	CheckConnectionMsg : STRING(255);
	PositionMsg : STRING(255);
	PositionCountMsg : STRING(255);
	IdMsg : STRING(255);
	CustomMsg : STRING(255);
	
	{region 'Commands'}
		
	{attribute 'OPC.UA.DA' := '0'}
	_moveAbsPosition     : BOOL;
	{attribute 'OPC.UA.DA' := '0'}
	_jogBackwardPosition : BOOL;
	{attribute 'OPC.UA.DA' := '0'}
	_jogForwardPosition  : BOOL;
	{attribute 'OPC.UA.DA' := '0'}
	_customCmd : BOOL;	
	
	{endregion}
	
	{attribute 'OPC.UA.DA' := '0'}
	_initDevice : BOOL;	
	
	{attribute 'OPC.UA.DA' := '0'}
	_pos : INT;	 
	{attribute 'OPC.UA.DA' := '0'}
	_cmd : STRING;	
	{attribute 'OPC.UA.DA' := '0'}
	_itemScheduler : INT;		
	{attribute 'OPC.UA.DA' := '0'}
	_pulseGenerator : TON;	
			
	{attribute 'OPC.UA.DA' := '0'}
	message : STRING;
	{attribute 'OPC.UA.DA' := '0'}
	_length : INT;
	
END_VAR


IF NOT InitConfigSerialCom THEN
	ConfigureSerialCom();
ELSE
	IF _refSerialCom.ErrorReceiveId = COMERROR_NOERROR THEN
		_refSerialCom(TxBuffer := HardwareGlobalVariables.TxBufferPolarisation, 
		 	      	  RxBuffer := HardwareGlobalVariables.RxBufferPolarisation);
	END_IF	
				  
	// Init device
	InitDevice(); 				  
				  
	// Deliver messages
	IF _refSerialCom.IsReceived THEN
		CASE _deliverMessages OF			
			EFeedbackMsgPolarisationFW212C.CheckConnectionMsg :
				CheckConnectionMsg := _refSerialCom.LastReceivedString;	
			EFeedbackMsgPolarisationFW212C.PositionMsg :
				PositionMsg := _refSerialCom.LastReceivedString;
			EFeedbackMsgPolarisationFW212C.PositionCountMsg :
				PositionCountMsg := _refSerialCom.LastReceivedString;
			EFeedbackMsgPolarisationFW212C.IdMsg :
				IdMsg := _refSerialCom.LastReceivedString;
			EFeedbackMsgPolarisationFW212C.CustomMsg :
				CustomMsg := _refSerialCom.LastReceivedString;						
		END_CASE
		
		_deliverMessages := 0;
	END_IF							   							   		
END_IF

IF InitConfigSerialCom THEN			
	MoveAbsPosition(_moveAbsPosition, _pos);	
	JogBackwardPosition(_jogBackwardPosition);				
	JogForwardPosition(_jogForwardPosition);
	CustomCommand(_customCmd, _cmd);	

	IF (NOT _moveAbsPosition AND NOT _jogBackwardPosition AND NOT _jogForwardPosition AND NOT _customCmd) THEN
		MessageScheduler();
	END_IF	
END_IF

METHOD CheckConnection
VAR_INPUT
END_VAR
VAR
	cmd : STRING := '';
END_VAR
_deliverMessages := EFeedbackMsgPolarisationFW212C.CheckConnectionMsg;
_serialCom.Send(cmd);
END_METHOD

METHOD ConfigureSerialCom
VAR_INPUT
END_VAR
IF _coeAccess.CoeOperation.Ready THEN
	_logger.Information(_message.Reset().Append('Start configuration com serial').ToString());
END_IF;	

_coeAccess.CoeOperation.Start();
_coeAccess(SerialCommunication := _config.SerialCommunication);
	
IF _coeAccess.CoeOperation.Done THEN
	_coeAccess.SetDone();
	
	_Logger.Information(_message.Reset().
							Append('{').Append(TO_STRING(THIS^.Family)).Append('} : ').
							Append(' - Status : ').Append(TO_STRING(_coeAccess.Status)).ToString());	
	InitConfigSerialCom := TRUE;
END_IF
 
IF _coeAccess.CoeOperation.Error THEN	
	_coeAccess.SetError(0);
	
	_Logger.Error(_message.Reset().
							Append('{').Append(TO_STRING(THIS^.Family)).Append('} : ').
							Append(' - Status : ').Append(TO_STRING(_coeAccess.Status)).ToString());	
	InitConfigSerialCom := TRUE;
END_IF

THIS^.Status := _coeAccess.Status;
State := _coeAccess.Status;
END_METHOD

{attribute 'TcRpcEnable' := '1'}
METHOD CustomCommand
VAR_INPUT
	Execute : BOOL;
	Cmd : STRING;
END_VAR
IF Execute THEN
	_logger.Information(_message.Reset().
								Append(_config.Name).
								Append(' - Custom : ').
								Append(Cmd).ToString());	
	_deliverMessages := EFeedbackMsgPolarisationFW212C.CustomMsg;								
	_serialCom.Send(Cmd);
	
	_customCmd := FALSE;
END_IF
END_METHOD

METHOD FB_init : BOOL
VAR_INPUT
	bInitRetains : BOOL; // if TRUE, the retain variables are initialized (warm start / cold start)
	bInCopyCode : BOOL;  // if TRUE, the instance afterwards gets moved into the copy code (online change)
	Config : FW212CPolarisationFilterConfig;
END_VAR
IF Config.IsEnabled THEN
	_config := Config;
	
	SUPER^._polarisationFilterConfig.Name := Config.Name;
	SUPER^._polarisationFilterConfig.DeviceID := Config.DeviceID;
	SUPER^._polarisationFilterConfig.IsEnabled := Config.IsEnabled;
	SUPER^._polarisationFilterConfig.LogLevel := Config.LogLevel;
	
	SUPER^.Name := Config.Name;
	SUPER^.DeviceID := Config.DeviceID;	
	THIS^.Family := DeviceFamily.PolarisationFilter;
	
	_Logger.Information(_message.Reset().Append('Init ').
							Append('{').Append(TO_STRING(THIS^.Family)).Append('} - ').
							Append('{').Append(TO_STRING(Config.Name)).Append('}').ToString());																													
END_IF
END_METHOD

(** Returns the model number and firmware version **)
METHOD GetIdentifier : STRING
VAR_INPUT
END_VAR
VAR
	cmd : STRING := '*idn?';
END_VAR
_deliverMessages := EFeedbackMsgPolarisationFW212C.IdMsg;
_serialCom.Send(cmd);
END_METHOD

(** Position Query **)
METHOD PROTECTED GetPosition 
VAR_INPUT
END_VAR
VAR
	cmd : STRING := 'pos?';
END_VAR
_deliverMessages := EFeedbackMsgPolarisationFW212C.PositionMsg;
_serialCom.Send(cmd);
END_METHOD

(** Returns the wheel type **)
METHOD GetPositionCount
VAR_INPUT
END_VAR
VAR
	cmd : STRING := 'pcount?';
END_VAR
_deliverMessages := EFeedbackMsgPolarisationFW212C.PositionCountMsg;
_serialCom.Send(cmd);
END_METHOD

PROPERTY InitConfigSerialCom : BOOL
GET
InitConfigSerialCom := _initConfigSerialCom;
END_GET
SET
_initConfigSerialCom := InitConfigSerialCom;
END_SET
END_PROPERTY

METHOD InitDevice
VAR_INPUT
END_VAR
IF NOT _initDevice THEN	
	_logger.Information(_message.Reset().
								Append(_config.Name).
								Append(' - Init device').ToString());

	// TODO : define max count 
	
	_initDevice := TRUE;	
END_IF
END_METHOD

{attribute 'TcRpcEnable' := '1'}
(** Decrements the filter position by 1 **)
METHOD PROTECTED JogBackwardPosition
VAR_INPUT
	Execute : BOOL;
END_VAR
VAR
	DecFilterPos : BYTE := 68;
	posArray     : ARRAY[1..3] OF BYTE := [27, 91, DecFilterPos];
END_VAR
IF Execute THEN
	_logger.Information(_message.Reset().
								Append(_config.Name).
								Append(' - Jog backward position').ToString());
	_serialCom.Send3B(posArray);
	_jogBackwardPosition := FALSE;
END_IF
END_METHOD

{attribute 'TcRpcEnable' := '1'}
(** Increments the filter position by 1 **)
METHOD PROTECTED JogForwardPosition
VAR_INPUT
	Execute : BOOL;
END_VAR
VAR
	jogForwardPos : BYTE := 67;
	posArray     : ARRAY[1..3] OF BYTE := [27, 91, jogForwardPos];
END_VAR
IF Execute THEN
	_logger.Information(_message.Reset().
								Append(_config.Name).
								Append(' - Jog forward position').ToString());
	_serialCom.Send3B(posArray);
	_jogForwardPosition := FALSE;
END_IF
END_METHOD

METHOD MessageScheduler
VAR_INPUT
END_VAR
IF _pulseGenerator.Q THEN
	_pulseGenerator(IN := FALSE, PT := T#10MS);
		
	CASE _itemScheduler OF
		0:  GetIdentifier();
			_itemScheduler := 1;

		1:	GetPosition();
			_itemScheduler := 2;
			
		2:  GetPositionCount();
			_itemScheduler := 3;
			
		3:  CheckConnection();
			_itemScheduler := 0;								
	END_CASE
ELSE
	_pulseGenerator(IN := TRUE, PT := T#50MS);	
END_IF
END_METHOD

{attribute 'TcRpcEnable' := '1'}
(** Moves the wheel to filter position n **)
METHOD PROTECTED MoveAbsPosition
VAR_INPUT
	Execute : BOOL;
	Position : LREAL;
END_VAR
VAR
	cmd : STRING := 'pos=';
END_VAR
IF Execute THEN
	_logger.Information(_message.Reset().
								Append(_config.Name).
								Append(' - Move absolute position : ').Append(TO_STRING(Position)).ToString());
	_serialCom.Send(CONCAT(cmd, TO_STRING(Position)));
	_moveAbsPosition := FALSE;
END_IF
END_METHOD

{attribute 'TcRpcEnable' := '1'}
METHOD RaisePropertiesChanged
VAR_INPUT
	Execute : BOOL;
END_VAR
IF Execute THEN
	CheckConnectionMsg := ' ';
	PositionMsg := ' ';
	IdMsg := ' ';
	CustomMsg := ' ';
END_IF
END_METHOD

END_FUNCTION_BLOCK

// ---- PMShared/Hardware/Devices/PolarisationFilters/PolarisationFilterBase.TcPOU
FUNCTION_BLOCK ABSTRACT PolarisationFilterBase EXTENDS TExecution IMPLEMENTS IDevice
VAR_INPUT
END_VAR
VAR_OUTPUT
END_VAR
VAR
	{attribute 'OPC.UA.DA' := '0'}
	_name : STRING;
	{attribute 'OPC.UA.DA' := '0'}
	_deviceID : STRING;					
	{attribute 'OPC.UA.DA' := '0'}
	_family : DeviceFamily;			
	{attribute 'OPC.UA.DA' := '0'}
	_logger : Logger;
	{attribute 'OPC.UA.DA' := '0'}
	_message : StringBuilder;
	{attribute 'OPC.UA.DA' := '0'}
	_polarisationFilterConfig : DeviceConfiguration;
END_VAR

PROPERTY DeviceID : STRING
GET
DeviceID := _deviceID;
END_GET
SET
_deviceID := DeviceID;
END_SET
END_PROPERTY

PROPERTY Family : DeviceFamily
GET
Family := _family;
END_GET
SET
_family := Family;
END_SET
END_PROPERTY

METHOD PROTECTED ABSTRACT GetPosition 
VAR_INPUT
END_VAR
END_METHOD

METHOD PROTECTED ABSTRACT JogBackwardPosition
VAR_INPUT
	Execute : BOOL;
END_VAR
END_METHOD

METHOD PROTECTED ABSTRACT JogForwardPosition
VAR_INPUT
	Execute : BOOL;
END_VAR
END_METHOD

METHOD PROTECTED ABSTRACT MoveAbsPosition
VAR_INPUT
	Execute : BOOL;
	Position : LREAL;
END_VAR
END_METHOD

PROPERTY Name : STRING
GET
Name := _name;
END_GET
SET
_name := Name;
END_SET
END_PROPERTY

END_FUNCTION_BLOCK

// ---- PMShared/Hardware/Devices/PolarisationFilters/Thorlabs/ELL14KPolarisationFilter.TcPOU
{attribute 'OPC.UA.DA' := '1'}
FUNCTION_BLOCK ELL14KPolarisationFilter EXTENDS PolarisationFilterBase
VAR_INPUT
END_VAR
VAR_OUTPUT
END_VAR
VAR
	{attribute 'OPC.UA.DA' := '0'}
	_config : ELL14KPolarisationFilterConfig;
	{attribute 'OPC.UA.DA' := '0'}
	_hsPolarisationConfig : PolarisationConfig;
	{attribute 'OPC.UA.DA' := '0'}
	_htPolarisationConfig : PolarisationConfig;
	{attribute 'OPC.UA.DA' := '0'}
	_coeAccess : CoeAccess;
	{attribute 'OPC.UA.DA' := '0'}
	_initConfigSerialCom : BOOL;	
	{attribute 'OPC.UA.DA' := '0'}
	_serialCom  : SerialCom(Prefix :='', Suffix := Const.CR_LF);
	{attribute 'OPC.UA.DA' := '0'}
	_refSerialCom : REFERENCE TO SerialCom(Prefix :='', Suffix := Const.CR_LF) := _serialCom;	 
	{attribute 'OPC.UA.DA' := '0'}
	_isReceived : BOOL;
	
	{attribute 'OPC.UA.DA' := '0'}
	_deliverMessages : INT;
	
	PositionMsg : STRING(255);
	IdMsg : STRING(255);
	CalibMsg : STRING(255);
	CustomMsg : STRING(255);
	
	{region 'Commands'}	
	
	{attribute 'OPC.UA.DA' := '0'}
	_homePosition 		: BOOL;
	{attribute 'OPC.UA.DA' := '0'}
	_moveAbsPosition	: BOOL;
	{attribute 'OPC.UA.DA' := '0'}
	_moveRelPosition	: BOOL;
	{attribute 'OPC.UA.DA' := '0'}
	_jogBackwardPosition : BOOL;
	{attribute 'OPC.UA.DA' := '0'}
	_jogForwardPosition  : BOOL;
	{attribute 'OPC.UA.DA' := '0'}
	_customCmd : BOOL;
	{attribute 'OPC.UA.DA' := '0'}			  		   
	_raiseProperties : BOOL;
	 		 
	{endregion}
	
	{attribute 'OPC.UA.DA' := '0'}
	_initDevice : BOOL;	
	{attribute 'OPC.UA.DA' := '0'}
	_polarResult : EPolar;
 	
	{attribute 'OPC.UA.DA' := '0'}
	_pos : LREAL;
	{attribute 'OPC.UA.DA' := '0'}
	_cmd : STRING;	
	{attribute 'OPC.UA.DA' := '0'}
	_itemScheduler : INT;	
	{attribute 'OPC.UA.DA' := '0'}
	_itemRaisedProperties : INT;		
	{attribute 'OPC.UA.DA' := '0'}
	_pulseGenerator : TON;	
			
	{attribute 'OPC.UA.DA' := '0'}
	tmpMessage : STRING;
	{attribute 'OPC.UA.DA' := '0'}
	message : STRING;
	{attribute 'OPC.UA.DA' := '0'}
	_length : INT;		 
	{attribute 'OPC.UA.DA' := '0'}
	_findSuffix : INT;
	{attribute 'OPC.UA.DA' := '0'}
	_roundPosition : STRING; 
	{attribute 'OPC.UA.DA' := '0'}
	hsS_temp : STRING;
	{attribute 'OPC.UA.DA' := '0'}
	hsP_temp : STRING;
	{attribute 'OPC.UA.DA' := '0'}
	htS_temp : STRING;
	{attribute 'OPC.UA.DA' := '0'}
	htP_temp : STRING;
	
	_delimeter : STRING := ';';
	{attribute 'OPC.UA.DA' := '0'}
	_firstConcat : STRING;
	{attribute 'OPC.UA.DA' := '0'}
	_secondConcat : STRING;
	{attribute 'OPC.UA.DA' := '0'}
	_thirdConcat : STRING;
	{attribute 'OPC.UA.DA' := '0'}
	_fourthConcat : STRING;
	{attribute 'OPC.UA.DA' := '0'}
	_fithConcat : STRING;
	{attribute 'OPC.UA.DA' := '0'}
	_sixthConcat : STRING;
	
END_VAR


IF NOT InitConfigSerialCom THEN
	ConfigureSerialCom();
ELSIF THIS^.Status = TExecutionState.Ready THEN
	IF _refSerialCom.ErrorReceiveId = COMERROR_NOERROR THEN
		_refSerialCom(TxBuffer:= HardwareGlobalVariables.TxBufferPolarisation, 
		 	          RxBuffer:= HardwareGlobalVariables.RxBufferPolarisation);
	END_IF	
				  
	// Init device
	InitDevice(); 				  
				  
	// Deliver messages
	IF _refSerialCom.IsReceived THEN
		CASE _deliverMessages OF			
			EFeedbackMsgPolarisationELL14K.PositionMsg :
				tmpMessage := DELETE(_refSerialCom.LastReceivedString, 3, 1);
				_length := LEN(tmpMessage);
				_findSuffix := FIND(tmpMessage, Const.CR_LF);
				message := DELETE(tmpMessage, 4, _findSuffix);
				
				PositionMsg := ConvertPulsesToDegrees(message);
				
				_roundPosition := LREAL_TO_FMTSTR(STRING_TO_LREAL(PositionMsg), 1, TRUE);	
				hsS_temp := LREAL_TO_FMTSTR(_hsPolarisationConfig.PolarAngle_S, 1, FALSE); 
				hsP_temp := LREAL_TO_FMTSTR(_hsPolarisationConfig.PolarAngle_P, 1, FALSE);
				htS_temp := LREAL_TO_FMTSTR(_htPolarisationConfig.PolarAngle_S, 1, FALSE); 
				htP_temp := LREAL_TO_FMTSTR(_htPolarisationConfig.PolarAngle_P, 1, FALSE);
				IF (_roundPosition = hsS_temp OR _roundPosition = htS_temp) THEN
					PolarResult := EPolar.S_Polar;
				ELSIF (_roundPosition = hsP_temp OR _roundPosition = htP_temp) THEN
					PolarResult := EPolar.P_Polar;		
				END_IF
								
				_logger.Information(_message.Reset().Append('ELL14KPolarisationFilter position: ').Append(PositionMsg).ToString());
				
			EFeedbackMsgPolarisationELL14K.IdMsg :
				IdMsg := _refSerialCom.LastReceivedString;							
			EFeedbackMsgPolarisationELL14K.CustomMsg :
				CustomMsg := _refSerialCom.LastReceivedString;						
		END_CASE
	ELSE
		CASE _deliverMessages OF
			EFeedbackMsgPolarisationELL14K.CalibMsg :
				_firstConcat := CONCAT(LREAL_TO_FMTSTR(_hsPolarisationConfig.PolarAngle_S, 1, FALSE), _delimeter);	
				_secondConcat := CONCAT(_firstConcat, LREAL_TO_FMTSTR(_hsPolarisationConfig.PolarAngle_P, 1, FALSE));	
				_thirdConcat := CONCAT(_secondConcat, _delimeter);
				_fourthConcat := CONCAT(_thirdConcat, LREAL_TO_FMTSTR(_htPolarisationConfig.PolarAngle_S, 1, FALSE));
				_fithConcat := CONCAT(_fourthConcat, _delimeter);				
				_sixthConcat := CONCAT(_fithConcat, LREAL_TO_FMTSTR(_htPolarisationConfig.PolarAngle_P, 1, FALSE));
			
				CalibMsg := _sixthConcat;
				_deliverMessages := EFeedbackMsgPolarisationELL14K.PositionMsg;
		END_CASE			
	END_IF							   	


	HomePosition(_homePosition);	
	MoveAbsPosition(_moveAbsPosition, _pos);
	MoveRelPosition(_moveRelPosition, _pos);	
	JogBackwardPosition(_jogBackwardPosition);				
	JogForwardPosition(_jogForwardPosition);
	CustomCommand(_customCmd, _cmd);		
	RaisePropertiesChanged(_raiseProperties);		
END_IF

METHOD ConfigureSerialCom
VAR_INPUT
END_VAR
IF _coeAccess.CoeOperation.Ready THEN
	_logger.Information(_message.Reset().Append('Start configuration com serial').ToString());
END_IF;	

_coeAccess.CoeOperation.Start();
_coeAccess(SerialCommunication := _config.SerialCommunication);
	
IF _coeAccess.CoeOperation.Done THEN
	_coeAccess.SetDone();	
 
	_Logger.Information(_message.Reset().
							Append('{').Append(TO_STRING(THIS^.Family)).Append('} : ').
							Append(' - Status : ').Append(TO_STRING(_coeAccess.Status)).ToString());	
	InitConfigSerialCom := TRUE;
END_IF
 
IF _coeAccess.CoeOperation.Error THEN	
	_coeAccess.SetError(0);
	
	_Logger.Error(_message.Reset().
							Append('{').Append(TO_STRING(THIS^.Family)).Append('} : ').
							Append(' - Status : ').Append(TO_STRING(_coeAccess.Status)).ToString());
	InitConfigSerialCom := TRUE;
END_IF

THIS^.Status := _coeAccess.Status;
State := _coeAccess.Status;
END_METHOD

METHOD ConvertDegreesToPulses : STRING
VAR_INPUT
	AnglePosition : LREAL;
END_VAR
VAR
	NumberPulses : DWORD;
END_VAR
NumberPulses := LREAL_TO_DWORD(AnglePosition * Const.PULSES_PER_DEG);	
ConvertDegreesToPulses := DWORD_TO_HEXSTR(NumberPulses, 8, FALSE );
END_METHOD

METHOD ConvertPulsesToDegrees : STRING
VAR_INPUT
	Pulses : STRING;
END_VAR
VAR
	pulsesInHex : STRING; 
	pulsesToDint : DINT;
END_VAR
pulsesInHex := CONCAT('16#', Pulses);
pulsesToDint := STRING_TO_DINT(pulsesInHex);
ConvertPulsesToDegrees := LREAL_TO_FMTSTR(ABS(DINT_TO_LREAL(pulsesToDint) / Const.PULSES_PER_DEG), 4, TRUE);
END_METHOD

{attribute 'TcRpcEnable' := '1'}
METHOD CustomCommand
VAR_INPUT
	Execute : BOOL;
	Cmd : STRING;
END_VAR
IF Execute THEN
	_logger.Information(_message.Reset().
								Append(_config.Name).
								Append(' - Custom : ').
								Append(Cmd).ToString());
	_deliverMessages := EFeedbackMsgPolarisationELL14K.CustomMsg;									
	_serialCom.Send(Cmd);
	
	_customCmd := FALSE;
END_IF
END_METHOD

METHOD FB_init : BOOL
VAR_INPUT
	bInitRetains : BOOL; // if TRUE, the retain variables are initialized (warm start / cold start)
	bInCopyCode : BOOL;  // if TRUE, the instance afterwards gets moved into the copy code (online change)
	Config : ELL14KPolarisationFilterConfig;
	HsPolarisationConfig : PolarisationConfig;
	HtPolarisationConfig : PolarisationConfig;
END_VAR
IF Config.IsEnabled THEN
	_config := Config;
	_hsPolarisationConfig := HsPolarisationConfig;
	_htPolarisationConfig := HtPolarisationConfig;
	
	SUPER^._polarisationFilterConfig.Name := Config.Name;
	SUPER^._polarisationFilterConfig.DeviceID := Config.DeviceID;
	SUPER^._polarisationFilterConfig.IsEnabled := Config.IsEnabled;
	SUPER^._polarisationFilterConfig.LogLevel := Config.LogLevel;
	
	SUPER^.Name := Config.Name;
	SUPER^.DeviceID := Config.DeviceID;	
	THIS^.Family := DeviceFamily.PolarisationFilter;
	
	_Logger.Information(_message.Reset().Append('Init ').
							Append('{').Append(TO_STRING(THIS^.Family)).Append('} - ').
							Append('{').Append(TO_STRING(Config.Name)).Append('}').ToString());																													
END_IF
END_METHOD

METHOD PROTECTED GetCalibConfig
VAR_INPUT
END_VAR
VAR
	
END_VAR
_deliverMessages := EFeedbackMsgPolarisationELL14K.CalibMsg;
END_METHOD

(** Returns the model number and firmware version **)
METHOD GetIdentifier
VAR_INPUT
END_VAR
VAR
	cmd : STRING := '0i1';
END_VAR
_deliverMessages := EFeedbackMsgPolarisationELL14K.IdMsg;	
_serialCom.Send(cmd);
END_METHOD

METHOD PROTECTED GetPosition
VAR_INPUT
END_VAR
VAR
	cmd : STRING := '0gp';
END_VAR
_deliverMessages := EFeedbackMsgPolarisationELL14K.PositionMsg;
_serialCom.Send(cmd);
END_METHOD

{attribute 'TcRpcEnable' := '1'}
METHOD HomePosition
VAR_INPUT
	Execute : BOOL;
END_VAR
VAR
	cmd : STRING := '0ho1';
END_VAR
IF Execute THEN
	_logger.Information(_message.Reset().
								Append(_config.Name).
								Append(' - Home position : ').ToString());
	
	PolarResult := EPolar.Unknown;
	
	_serialCom.Send(cmd);	
	_homePosition := FALSE;
END_IF
END_METHOD

PROPERTY InitConfigSerialCom : BOOL
GET
InitConfigSerialCom := _initConfigSerialCom;
END_GET
SET
_initConfigSerialCom := InitConfigSerialCom;
END_SET
END_PROPERTY

METHOD InitDevice
VAR_INPUT
END_VAR
IF NOT _initDevice THEN	
	_logger.Information(_message.Reset().
								Append(_config.Name).
								Append(' - Init device').ToString());	
	_initDevice := TRUE;
	//_raiseProperties := TRUE;
	
	GetPosition();	
END_IF
END_METHOD

{attribute 'TcRpcEnable' := '1'}
METHOD PROTECTED JogBackwardPosition
VAR_INPUT
	Execute : BOOL;
END_VAR
VAR
	cmd : STRING := '0bw';
END_VAR
IF Execute THEN
	_logger.Information(_message.Reset().
								Append(_config.Name).
								Append(' - Jog backward position : ').ToString());
	_serialCom.Send(cmd);
	
	_jogBackwardPosition := FALSE;
END_IF
END_METHOD

{attribute 'TcRpcEnable' := '1'}
METHOD PROTECTED JogForwardPosition
VAR_INPUT
	Execute : BOOL;
END_VAR
VAR
	cmd : STRING := '0fw';
END_VAR
IF Execute THEN
	_logger.Information(_message.Reset().
								Append(_config.Name).
								Append(' - Jog forward position : ').ToString());
	_serialCom.Send(cmd);
	
	_jogForwardPosition := FALSE;
END_IF
END_METHOD

{attribute 'TcRpcEnable' := '1'}
METHOD PROTECTED MoveAbsPosition 
VAR_INPUT
	Execute : BOOL;
	Position : LREAL;
END_VAR
VAR
	cmd : STRING := '0ma';
END_VAR
IF Execute THEN
	_pos := Position;	

	_logger.Information(_message.Reset().
								Append(_config.Name).
								Append(' - Move absolute position : ').Append(TO_STRING(_pos)).ToString());
		
	PolarResult := EPolar.Unknown;					
								
	_serialCom.Send(CONCAT(cmd, ConvertDegreesToPulses(_pos)));
	_moveAbsPosition := FALSE;	
END_IF
END_METHOD

{attribute 'TcRpcEnable' := '1'}
METHOD PROTECTED MoveRelPosition 
VAR_INPUT
	Execute : BOOL;
	AnglePosition : LREAL;
END_VAR
VAR
	cmd : STRING := '0mr';
END_VAR
IF Execute THEN
	_pos := AnglePosition;	
	_logger.Information(_message.Reset().
								Append(_config.Name).
								Append(' - Move relative position : ').Append(TO_STRING(_pos)).ToString());
	
	PolarResult := EPolar.Unknown;
	
	_serialCom.Send(CONCAT(cmd, ConvertDegreesToPulses(_pos)));	
	_moveRelPosition := FALSE;
END_IF
END_METHOD

PROPERTY PUBLIC PolarResult : EPolar
GET
PolarResult := _polarResult;
END_GET
SET
_polarResult := PolarResult;
END_SET
END_PROPERTY

{attribute 'TcRpcEnable' := '1'}
METHOD RaisePropertiesChanged
VAR_INPUT
	Execute : BOOL;
END_VAR
IF Execute THEN
	IF THIS^.Status <> TExecutionState.Ready THEN	
		_raiseProperties := FALSE;
		RETURN;
	END_IF
	
	_raiseProperties := TRUE;
	
	IF _pulseGenerator.Q THEN
		_pulseGenerator(IN := FALSE, PT := T#10MS);	

		CASE _itemRaisedProperties OF
			0:  PositionMsg := ' ';
				IdMsg := ' ';
				CalibMsg := ' ';
				CustomMsg := ' ';
				
				_itemRaisedProperties := 10;
			
			10:  GetIdentifier();
				_itemRaisedProperties := 11;
				
			11:  GetPosition();
				_itemRaisedProperties := 12;
				
			12: GetCalibConfig();
				_itemRaisedProperties := 20;
			
			20:  _logger.Information(_message.Reset().
								Append(_config.Name).
								Append(' - Polarisation RaisePropertiesChanged').ToString());
				_raiseProperties := FALSE;				
				_itemRaisedProperties := 0;
			
		END_CASE
	ELSE
		_pulseGenerator(IN := TRUE, PT := T#100MS);	
	END_IF
END_IF
END_METHOD

END_FUNCTION_BLOCK

// ---- PMShared/Hardware/Devices/Lasers/Quantum/SMD12Laser.TcPOU
{attribute 'OPC.UA.DA' := '1'}
FUNCTION_BLOCK SMD12Laser EXTENDS LaserBase
VAR_INPUT
END_VAR
VAR_OUTPUT
END_VAR
VAR
	{attribute 'OPC.UA.DA' := '0'}
	_config : SMD12LaserConfig;	
	{attribute 'OPC.UA.DA' := '0'}
	_coeAccess : CoeAccess;	
	{attribute 'OPC.UA.DA' := '0'}
	_initConfigSerialCom : BOOL;	
	{attribute 'OPC.UA.DA' := '0'}
	_serialCom  : SerialCom(Prefix :='', Suffix := Const.CARRIAGE_RETURN);
	{attribute 'OPC.UA.DA' := '0'}
	_refSerialCom : REFERENCE TO SerialCom(Prefix :='', Suffix := Const.CARRIAGE_RETURN) := _serialCom;		 
	{attribute 'OPC.UA.DA' := '0'}
	_isReceived : BOOL;
	
	{attribute 'OPC.UA.DA' := '0'}
	_deliverMessages : INT;
	
	PowerMsg : STRING(255);
	InterlockStatusMsg : STRING(255);
	LaserTemperatureMsg : STRING(255);
	PsuTemperatureMsg : STRING(255);
	IdMsg : STRING(255);
	CustomMsg : STRING(255);
	
	{region 'Commands'}
	
	{attribute 'OPC.UA.DA' := '0'}
	_powerOn : BOOL;
	{attribute 'OPC.UA.DA' := '0'}
	_powerOff : BOOL;
	{attribute 'OPC.UA.DA' := '0'}
	_setPowerCmd : BOOL;
	{attribute 'OPC.UA.DA' := '0'}	 
	_setCurrentCmd : BOOL;
	{attribute 'OPC.UA.DA' := '0'}			 
	_controlModeCmd : BOOL;
	{attribute 'OPC.UA.DA' := '0'}
	_customCmd : BOOL;	
	{attribute 'OPC.UA.DA' := '0'}			  		   
	_raiseProperties : BOOL;
	
	{endregion}			
	
	{attribute 'OPC.UA.DA' := '0'}
	_initDevice : BOOL;	
	 
	{attribute 'OPC.UA.DA' := '0'}
	_cmd : STRING;			
	{attribute 'OPC.UA.DA' := '0'}
	_setpoint : LREAL := 0;
	{attribute 'OPC.UA.DA' := '0'}
	_itemScheduler : INT;
	{attribute 'OPC.UA.DA' := '0'}
	_itemExecScheduler : INT;		
	{attribute 'OPC.UA.DA' := '0'}
	_itemRaisedProperties : INT;			
	{attribute 'OPC.UA.DA' := '0'}
	_pulseGenerator : TON;	
	{attribute 'OPC.UA.DA' := '0'}
	_execPulseGenerator : TON;	
			
	{attribute 'OPC.UA.DA' := '0'}
	message : STRING;
	{attribute 'OPC.UA.DA' := '0'}	
	_length : INT;
	{attribute 'OPC.UA.DA' := '0'}
	_mode : EControlModeSmd12;	
END_VAR

IF NOT InitConfigSerialCom THEN
	ConfigureSerialCom();
ELSIF THIS^.Status = TExecutionState.Ready THEN
	IF _refSerialCom.ErrorReceiveId = COMERROR_NOERROR THEN
		_refSerialCom(TxBuffer:= HardwareGlobalVariables.TxBufferLaser, 
		 	      	  RxBuffer:= HardwareGlobalVariables.RxBufferLaser);
	END_IF				  
	
	// Init device
	InitDevice(); 				  				 

	// Deliver messages
	IF _refSerialCom.IsReceived THEN				 	
		CASE _deliverMessages OF			
			EFeedbackMsgSMD12.PowerMsg :		
				message := DELETE(_refSerialCom.LastReceivedString, 3, 0);
				_length := LEN(message);		
				PowerMsg := DELETE(message, 4, _length-2);		
			EFeedbackMsgSMD12.InterlockStatusMsg :
				message := DELETE(_refSerialCom.LastReceivedString, 2, 0);
				_length := LEN(message);	
				InterlockStatusMsg := DELETE(message, 2, _length);
			EFeedbackMsgSMD12.LaserTemperatureMsg :
				message := DELETE(_refSerialCom.LastReceivedString, 3, 0);
				_length := LEN(message);		
				LaserTemperatureMsg := DELETE(message, 3, _length-1);
			EFeedbackMsgSMD12.PsuTemperatureMsg :
				message := DELETE(_refSerialCom.LastReceivedString, 3, 0);
				_length := LEN(message);		
				PsuTemperatureMsg := DELETE(message, 3, _length-1);
			EFeedbackMsgSMD12.IdMsg :
				message := DELETE(_refSerialCom.LastReceivedString, 3, 0);
				_length := LEN(message);		
				IdMsg := DELETE(message, 2, _length);
			EFeedbackMsgSMD12.CustomMsg :
				message := DELETE(_refSerialCom.LastReceivedString, 2, 0);
				_length := LEN(message);		
				CustomMsg := DELETE(message, 3, _length);
		END_CASE		
	END_IF								   							   	
	
	PowerOn(_powerOn);
	PowerOff(_powerOff);	
	ControlMode(_controlModeCmd, _mode); 
	SetPower(_setPowerCmd, _setpoint);
	SetCurrent(_setCurrentCmd, _setpoint);
	CustomCommand(_customCmd, _cmd);
	RaisePropertiesChanged(_raiseProperties);
	
	IF (NOT _powerOn AND NOT _powerOff AND NOT _controlModeCmd AND NOT _setPowerCmd AND NOT _setCurrentCmd 
		AND NOT _customCmd AND NOT _raiseProperties) THEN
		MessageScheduler();
	END_IF
END_IF

METHOD ConfigureSerialCom
VAR_INPUT
END_VAR
IF _coeAccess.CoeOperation.Ready THEN
	_logger.Information(_message.Reset().Append('Start configuration com serial').ToString());
END_IF;	

_coeAccess.CoeOperation.Start();
_coeAccess(SerialCommunication := _config.SerialCommunication);
	
IF _coeAccess.CoeOperation.Done THEN
	_coeAccess.SetDone();	
	
	_Logger.Information(_message.Reset().
							Append('{').Append(TO_STRING(THIS^.Family)).Append('} : ').
							Append(' - Status : ').Append(TO_STRING(_coeAccess.Status)).ToString());	
	InitConfigSerialCom := TRUE;
END_IF
 
IF _coeAccess.CoeOperation.Error THEN	
	_coeAccess.SetError(0);
	
	_Logger.Error(_message.Reset().
							Append('{').Append(TO_STRING(THIS^.Family)).Append('} : ').
							Append(' - Status : ').Append(TO_STRING(_coeAccess.Status)).ToString());
	InitConfigSerialCom := TRUE;
END_IF

THIS^.Status := _coeAccess.Status;
State := _coeAccess.Status;
END_METHOD

METHOD ControlMode
VAR_INPUT
	Execute : BOOL;
	Mode : EControlModeSmd12;
END_VAR
VAR
	currentModecmd : STRING := 'CONTROL=CURRENT';
	powerModecmd : STRING := 'CONTROL=POWER';
END_VAR
IF Execute THEN
	_logger.Information(_message.Reset().
								Append(_config.Name).
								Append(' - ControlMode : ').Append(TO_STRING(Mode)).ToString());
	
	IF MODE = EControlModeSmd12.CurrentMode THEN
		_serialCom.Send(currentModecmd);
	ELSIF MODE = EControlModeSmd12.PowerMode THEN
		_serialCom.Send(powerModecmd);
	END_IF
	
	_controlModeCmd := FALSE;		
END_IF
END_METHOD

{attribute 'TcRpcEnable' := '1'}
(** Custom command **)
METHOD CustomCommand
VAR_INPUT
	Execute : BOOL;
	Cmd : STRING;
END_VAR
IF Execute THEN
	_logger.Information(_message.Reset().
								Append(_config.Name).
								Append(' - Custom command : ').
								Append(Cmd).ToString());	
	_deliverMessages := EFeedbackMsgSMD12.CustomMsg;														
	_serialCom.Send(Cmd);	
	_customCmd := FALSE;
END_IF
END_METHOD

METHOD FB_init : BOOL
VAR_INPUT
	bInitRetains : BOOL; // if TRUE, the retain variables are initialized (warm start / cold start)
	bInCopyCode : BOOL;  // if TRUE, the instance afterwards gets moved into the copy code (online change)
	Config : SMD12LaserConfig;
END_VAR
IF Config.IsEnabled THEN
	_config := Config;
	
	SUPER^._laserConfig.Name := Config.Name;
	SUPER^._laserConfig.DeviceID := Config.DeviceID;
	SUPER^._laserConfig.IsEnabled := Config.IsEnabled;
	SUPER^._laserConfig.LogLevel := Config.LogLevel;
	
	SUPER^.Name := Config.Name;
	SUPER^.DeviceID := Config.DeviceID;	
	THIS^.Family := DeviceFamily.Laser;
		
	_Logger.Information(_message.Reset().Append('Init ').
							Append('{').Append(TO_STRING(THIS^.Family)).Append('} - ').
							Append('{').Append(TO_STRING(Config.Name)).Append('}').ToString());																													
END_IF
END_METHOD

METHOD GetIdentifier
VAR_INPUT
END_VAR
VAR
	cmd : STRING := 'VERSION?';
END_VAR
_deliverMessages := EFeedbackMsgSMD12.IdMsg;
_serialCom.Send(cmd);
END_METHOD

(** Returns the status of the Interlock **)
METHOD PROTECTED GetInterlockStatus 
VAR_INPUT
END_VAR
VAR
	cmd : STRING := 'STATUS?';
END_VAR
_deliverMessages := EFeedbackMsgSMD12.InterlockStatusMsg;
_serialCom.Send(cmd);
END_METHOD

(** Returns the temperature of the laser head in degrees centigrade **)
METHOD GetLaserTemperature 
VAR_INPUT
END_VAR
VAR
	cmd : STRING := 'LASTEMP?';
END_VAR
_deliverMessages := EFeedbackMsgSMD12.LaserTemperatureMsg;
_serialCom.Send(cmd);
END_METHOD

(** Returns the temperature of the PSU in degrees centigrade **)
METHOD GetPsuTemperature
VAR_INPUT
END_VAR
VAR
	cmd : STRING := 'PSUTEMP?';
END_VAR
_deliverMessages := EFeedbackMsgSMD12.PsuTemperatureMsg;
_serialCom.Send(cmd);
END_METHOD

{attribute 'TcRpcEnable' := '1'}
(** Returns the timers of the laser and PSU:
		PSU Time=#######.#     Total time the system has been powered
		Laser Enabled Time=#######.#     Total time the diodes have been powered
		Laser OperationTime=#######.#    Total time the diodes have been powered >1 A  
**)
METHOD GetTimers : HoursStruct
VAR_INPUT
	Execute : BOOL;
END_VAR
VAR
	cmd : STRING := 'TIMERS?';
END_VAR
IF Execute THEN
	_logger.Information(_message.Reset().
								Append(_config.Name).
								Append(' - GetTimers').ToString());
	_serialCom.Send(cmd);
END_IF
END_METHOD

PROPERTY InitConfigSerialCom : BOOL
GET
InitConfigSerialCom := _initConfigSerialCom;
END_GET
SET
_initConfigSerialCom := InitConfigSerialCom;
END_SET
END_PROPERTY

METHOD InitDevice
VAR_INPUT
END_VAR
IF NOT _initDevice THEN	
	_logger.Information(_message.Reset().
								Append(_config.Name).
								Append(' - InitDevice').ToString());	
	_raiseProperties:= TRUE;	
	_initDevice := TRUE;	
END_IF
END_METHOD

METHOD MessageScheduler
VAR_INPUT
END_VAR
IF _pulseGenerator.Q THEN
	_pulseGenerator(IN := FALSE, PT := T#10MS);
		
	CASE _itemScheduler OF		
		0:	ReadPower();
			_itemScheduler := 1;				
	
		1:  GetLaserTemperature();
			_itemScheduler := 2;	
		
		2:  GetPsuTemperature();
			_itemScheduler := 0;		
	END_CASE
ELSE
	_pulseGenerator(IN := TRUE, PT := T#100MS);		
END_IF
END_METHOD

{attribute 'TcRpcEnable' := '1'}
(** Disables the laser, regardless of the interlock status **)
METHOD PROTECTED PowerOff
VAR_INPUT
	Execute : BOOL;
END_VAR
VAR
	cmd : STRING := 'OFF';
END_VAR
IF Execute THEN	
	_powerOff := TRUE;	
	
	IF _execPulseGenerator.Q THEN
		_execPulseGenerator(IN := FALSE, PT := T#10MS);
			
		CASE _itemExecScheduler OF
			0: _logger.Information(_message.Reset().
								Append(_config.Name).
								Append(' - PowerOff').ToString());
				_serialCom.Send(cmd);
				_itemExecScheduler := 1;
			
			1:  GetInterlockStatus();
				_itemExecScheduler := 2;
				
			2:  _powerOff := FALSE;	
				_itemExecScheduler := 0;		
								
		END_CASE
	ELSE
		_execPulseGenerator(IN := TRUE, PT := T#100MS);	
	END_IF
END_IF
END_METHOD

{attribute 'TcRpcEnable' := '1'}
(* Enables the laser subject to Interlock and Enable Switch status *)
METHOD PROTECTED PowerOn
VAR_INPUT
	Execute : BOOL;
END_VAR
VAR
	cmd : STRING := 'ON';
END_VAR
IF Execute THEN	
	_powerOn := TRUE;	

	IF _execPulseGenerator.Q THEN
		_execPulseGenerator(IN := FALSE, PT := T#10MS);
			
		CASE _itemExecScheduler OF
			0: _logger.Information(_message.Reset().
								Append(_config.Name).
								Append(' - PowerOn').ToString());
				_serialCom.Send(cmd);
				_itemExecScheduler := 1;
			
			1:  GetInterlockStatus();
				_itemExecScheduler := 2;
				
			2:  _powerOn := FALSE;	
				_itemExecScheduler := 0;		
								
		END_CASE
	ELSE
		_execPulseGenerator(IN := TRUE, PT := T#100MS);	
	END_IF
END_IF
END_METHOD

{attribute 'TcRpcEnable' := '1'}
METHOD RaisePropertiesChanged
VAR_INPUT
	Execute : BOOL;
END_VAR
IF Execute THEN
	_raiseProperties := TRUE;
	
	IF _pulseGenerator.Q THEN
		_pulseGenerator(IN := FALSE, PT := T#10MS);	

		CASE _itemRaisedProperties OF
			0:  InterlockStatusMsg := ' ';
				IdMsg := ' ';
				CustomMsg := ' ';
				
				_itemRaisedProperties := 10;
			
			10:  GetIdentifier();
				_itemRaisedProperties := 11;
				
			11:  GetInterlockStatus();
				_itemRaisedProperties := 12;
			
			12:  _logger.Information(_message.Reset().
								Append(_config.Name).
								Append(' - RaisePropertiesChanged').ToString());
				_raiseProperties := FALSE;				
				_itemRaisedProperties := 0;
			
		END_CASE
	ELSE
		_pulseGenerator(IN := TRUE, PT := T#100MS);	
	END_IF
END_IF
END_METHOD

(** Returns the power of the laser **)
METHOD PROTECTED ReadPower 
VAR_INPUT
END_VAR
VAR
	cmd : STRING := 'POWER?';
END_VAR
_deliverMessages := EFeedbackMsgSMD12.PowerMsg;	
_serialCom.Send(cmd);
END_METHOD

{attribute 'TcRpcEnable' := '1'}
METHOD SetCurrent 
VAR_INPUT
	Execute : BOOL;
	Current : LREAL;
END_VAR
VAR
	cmd : STRING := 'CURRENT=';
END_VAR
IF Execute THEN	
	_setCurrentCmd := TRUE;	
	
	_setpoint := Current;

	IF _execPulseGenerator.Q THEN
		_execPulseGenerator(IN := FALSE, PT := T#10MS);
			
		CASE _itemExecScheduler OF
			0: _logger.Information(_message.Reset().
								Append(_config.Name).
								Append(' - SetCurrent : ').Append(TO_STRING(_setpoint)).ToString());
				_serialCom.Send(CONCAT(cmd, TO_STRING(_setpoint)));
				_itemExecScheduler := 1;
			
			1:  _setCurrentCmd := FALSE;	
				_itemExecScheduler := 0;		
								
		END_CASE
	ELSE
		_execPulseGenerator(IN := TRUE, PT := T#100MS);	
	END_IF
END_IF
END_METHOD

{attribute 'TcRpcEnable' := '1'}
(** This sets the output power of the laser 
For example, to set a power of 2800 mW, send the string POWER=2800, followed by striking the RETURN key
**)
METHOD PROTECTED SetPower 
VAR_INPUT
	Execute : BOOL;
	Power : LREAL;
END_VAR
VAR
	cmd : STRING := 'POWER=';
END_VAR
IF Execute THEN	
	_setPowerCmd := TRUE;	

	_setpoint := Power;
	
	IF _execPulseGenerator.Q THEN
		_execPulseGenerator(IN := FALSE, PT := T#10MS);
			
		CASE _itemExecScheduler OF
			0: _logger.Information(_message.Reset().
								Append(_config.Name).
								Append(' - SetPower : ').Append(TO_STRING(_setpoint)).ToString());
				_serialCom.Send(CONCAT(cmd, TO_STRING(_setpoint)));
				_itemExecScheduler := 1;
			
			1:  ReadPower();
				_itemExecScheduler := 2;
				
			2:  _setPowerCmd := FALSE;	
				_itemExecScheduler := 0;		
								
		END_CASE
	ELSE
		_execPulseGenerator(IN := TRUE, PT := T#100MS);	
	END_IF
END_IF
END_METHOD

END_FUNCTION_BLOCK

// ---- PMShared/Hardware/Devices/Lasers/LaserBase.TcPOU
FUNCTION_BLOCK ABSTRACT LaserBase EXTENDS TExecution IMPLEMENTS IDevice
VAR_INPUT
END_VAR
VAR_OUTPUT
END_VAR
VAR
	{attribute 'OPC.UA.DA' := '0'}
	_name : STRING;
	{attribute 'OPC.UA.DA' := '0'}
	_deviceID : STRING;				
	{attribute 'OPC.UA.DA' := '0'}	
	_family : DeviceFamily;	
	{attribute 'OPC.UA.DA' := '0'}
	_logger : Logger;
	{attribute 'OPC.UA.DA' := '0'}
	_message : StringBuilder;
	{attribute 'OPC.UA.DA' := '0'}
	_laserConfig : DeviceConfiguration;	
END_VAR

PROPERTY DeviceID : STRING
GET
DeviceID := _deviceID;
END_GET
SET
_deviceID := DeviceID;
END_SET
END_PROPERTY

PROPERTY Family : DeviceFamily
GET
Family := _family;
END_GET
SET
_family := Family;
END_SET
END_PROPERTY

METHOD PROTECTED ABSTRACT GetInterlockStatus 
VAR_INPUT
END_VAR
END_METHOD

PROPERTY Name : STRING
GET
Name := _name;
END_GET
SET
_name := Name;
END_SET
END_PROPERTY

METHOD PROTECTED ABSTRACT PowerOff
VAR_INPUT
	Execute : BOOL;
END_VAR
END_METHOD

METHOD PROTECTED ABSTRACT PowerOn
VAR_INPUT
	Execute : BOOL;
END_VAR
END_METHOD

METHOD PROTECTED ABSTRACT ReadPower 
VAR_INPUT
END_VAR
END_METHOD

METHOD PROTECTED ABSTRACT SetPower
VAR_INPUT
	Execute : BOOL;
	Power : LREAL;
END_VAR
END_METHOD

END_FUNCTION_BLOCK

// ---- PMShared/Hardware/Devices/Lasers/Coherent/Sapphire488Laser.TcPOU
{attribute 'OPC.UA.DA' := '1'}
FUNCTION_BLOCK Sapphire488Laser EXTENDS LaserBase
VAR_INPUT
END_VAR
VAR_OUTPUT
END_VAR
VAR
	{attribute 'OPC.UA.DA' := '0'}
	_config : Sapphire488LaserConfig;	
	{attribute 'OPC.UA.DA' := '0'}
	_coeAccess : CoeAccess;	
	{attribute 'OPC.UA.DA' := '0'}
	_initConfigSerialCom : BOOL;	
	{attribute 'OPC.UA.DA' := '0'}
	_suffix : STRING := Const.CR_LF;
	{attribute 'OPC.UA.DA' := '0'}
	_serialCom  : SerialCom(Prefix :='', Suffix := _suffix);
	{attribute 'OPC.UA.DA' := '0'}
	_refSerialCom : REFERENCE TO SerialCom(Prefix :='', Suffix := _suffix) := _serialCom;		 
	{attribute 'OPC.UA.DA' := '0'}
	_isReceived : BOOL;
	
	
	{attribute 'OPC.UA.DA' := '0'}
	_deliverMessages : INT;
	
	PowerMsg : STRING(255);
	InterlockStatusMsg : STRING(255);
	BasePlateTemperatureMsg : STRING(255);
	ControllerTemperatureMsg : STRING(255);
	DiodeSetTemperatureMsg : STRING(255);
	MeasuredTemperatureMsg : STRING(255);
	LaserHeadReachedDiodeCurrentLimitMsg : STRING(255);
	IdMsg : STRING(255);
	CustomMsg : STRING(255);
	
	{region 'Commands'}
	
	{attribute 'OPC.UA.DA' := '0'}
	_powerOn : BOOL;
	{attribute 'OPC.UA.DA' := '0'}
	_powerOff : BOOL;
	{attribute 'OPC.UA.DA' := '0'}
	_setPowerCmd : BOOL;
	{attribute 'OPC.UA.DA' := '0'}
	_customCmd : BOOL;	
	{attribute 'OPC.UA.DA' := '0'}			  		   
	_raiseProperties : BOOL;
	
	{endregion}			
	
	{attribute 'OPC.UA.DA' := '0'}
	_initDevice : BOOL;	
	 
	{attribute 'OPC.UA.DA' := '0'}
	_cmd : STRING;			
	{attribute 'OPC.UA.DA' := '0'}
	_setpoint : LREAL := 0;
	{attribute 'OPC.UA.DA' := '0'}
	_itemScheduler : INT;
	{attribute 'OPC.UA.DA' := '0'}
	_itemExecScheduler : INT;		
	{attribute 'OPC.UA.DA' := '0'}
	_itemRaisedProperties : INT;			
	{attribute 'OPC.UA.DA' := '0'}
	_pulseGenerator : TON;	
	{attribute 'OPC.UA.DA' := '0'}
	_execPulseGenerator : TON;	
			
	{attribute 'OPC.UA.DA' := '0'}
	fullMessage : STRING;
	{attribute 'OPC.UA.DA' := '0'}
	message : STRING;
	{attribute 'OPC.UA.DA' := '0'}	
	_length : INT;
	{attribute 'OPC.UA.DA' := '0'}	
	_suffixLength : INT := LEN(_suffix);	
END_VAR

IF NOT InitConfigSerialCom THEN
	ConfigureSerialCom();
ELSIF THIS^.Status = TExecutionState.Ready THEN
	IF _refSerialCom.ErrorReceiveId = COMERROR_NOERROR THEN
		_refSerialCom(TxBuffer:= HardwareGlobalVariables.TxBufferLaser, 
		 	      	  RxBuffer:= HardwareGlobalVariables.RxBufferLaser);
	END_IF				  
	
	// Init device
	IF NOT _initDevice THEN	
		InitDevice(); 		
	ELSE;
		// Deliver messages
		IF _refSerialCom.IsReceived THEN				 
			fullMessage := _refSerialCom.LastReceivedString;
			_length := LEN(fullMessage);
			message := DELETE(fullMessage, _suffixLength, _length-_suffixLength+1);
			
			CASE _deliverMessages OF			
				EFeedbackMsgSapphire488.PowerMsg :	
					PowerMsg := message;		
				EFeedbackMsgSapphire488.InterlockStatusMsg :
					InterlockStatusMsg := message;
				EFeedbackMsgSapphire488.BasePlateTemperatureMsg :
					BasePlateTemperatureMsg := message;
				EFeedbackMsgSapphire488.ControllerTemperatureMsg :
					ControllerTemperatureMsg := message;
				EFeedbackMsgSapphire488.DiodeSetTemperatureMsg :
					DiodeSetTemperatureMsg := message;
				EFeedbackMsgSapphire488.MeasuredTemperatureMsg :
					MeasuredTemperatureMsg := message;
				EFeedbackMsgSapphire488.LaserHeadReachedDiodeCurrentLimitMsg :
					LaserHeadReachedDiodeCurrentLimitMsg := message;
				EFeedbackMsgSapphire488.IdMsg :	
					IdMsg := message;
				EFeedbackMsgSapphire488.CustomMsg :
					CustomMsg := message;
			END_CASE		
		END_IF								   							   	
		
		PowerOn(_powerOn);
		PowerOff(_powerOff);	
		SetPower(_setPowerCmd, _setpoint);
		CustomCommand(_customCmd, _cmd);
		RaisePropertiesChanged(_raiseProperties);
		
		IF (NOT _powerOn AND NOT _powerOff AND NOT _setPowerCmd  
			AND NOT _customCmd AND NOT _raiseProperties) THEN
			MessageScheduler();
		END_IF
	
	END_IF
END_IF

METHOD ConfigureSerialCom
VAR_INPUT
END_VAR
IF _coeAccess.CoeOperation.Ready THEN
	_logger.Information(_message.Reset().Append('Start configuration com serial').ToString());
END_IF;	

_coeAccess.CoeOperation.Start();
_coeAccess(SerialCommunication := _config.SerialCommunication);
	
IF _coeAccess.CoeOperation.Done THEN
	_coeAccess.SetDone();	
	
	_Logger.Information(_message.Reset().
							Append('{').Append(TO_STRING(THIS^.Family)).Append('} : ').
							Append(' - Status : ').Append(TO_STRING(_coeAccess.Status)).ToString());	
	InitConfigSerialCom := TRUE;
END_IF
 
IF _coeAccess.CoeOperation.Error THEN	
	_coeAccess.SetError(0);
	
	_Logger.Error(_message.Reset().
							Append('{').Append(TO_STRING(THIS^.Family)).Append('} : ').
							Append(' - Status : ').Append(TO_STRING(_coeAccess.Status)).ToString());
	InitConfigSerialCom := TRUE;
END_IF

THIS^.Status := _coeAccess.Status;
State := _coeAccess.Status;
END_METHOD

{attribute 'TcRpcEnable' := '1'}
(** Custom command **)
METHOD CustomCommand
VAR_INPUT
	Execute : BOOL;
	Cmd : STRING;
END_VAR
IF Execute THEN
	_logger.Information(_message.Reset().
								Append(_config.Name).
								Append(' - Custom command : ').
								Append(Cmd).ToString());	
	_deliverMessages := EFeedbackMsgSapphire488.CustomMsg;														
	_serialCom.Send(Cmd);	
	_customCmd := FALSE;
END_IF
END_METHOD

METHOD FB_init : BOOL
VAR_INPUT
	bInitRetains : BOOL; // if TRUE, the retain variables are initialized (warm start / cold start)
	bInCopyCode : BOOL;  // if TRUE, the instance afterwards gets moved into the copy code (online change)
	Config : Sapphire488LaserConfig;
END_VAR
IF Config.IsEnabled THEN
	_config := Config;
	
	SUPER^._laserConfig.Name := Config.Name;
	SUPER^._laserConfig.DeviceID := Config.DeviceID;
	SUPER^._laserConfig.IsEnabled := Config.IsEnabled;
	SUPER^._laserConfig.LogLevel := Config.LogLevel;
	
	SUPER^.Name := Config.Name;
	SUPER^.DeviceID := Config.DeviceID;	
	THIS^.Family := DeviceFamily.Laser;
		
	_Logger.Information(_message.Reset().Append('Init ').
							Append('{').Append(TO_STRING(THIS^.Family)).Append('} - ').
							Append('{').Append(TO_STRING(Config.Name)).Append('}').ToString());																													
END_IF
END_METHOD

METHOD GetBasePlateTemperature 
VAR_INPUT
END_VAR
VAR
	cmd : STRING := '?BT';
END_VAR
_deliverMessages := EFeedbackMsgSapphire488.BasePlateTemperatureMsg;
_serialCom.Send(cmd);
END_METHOD

METHOD GetControllerTemperature
VAR_INPUT
END_VAR
VAR
	cmd : STRING := '?PST';
END_VAR
_deliverMessages := EFeedbackMsgSapphire488.ControllerTemperatureMsg;
_serialCom.Send(cmd);
END_METHOD

METHOD GetDiodeSetTemperature 
VAR_INPUT
END_VAR
VAR
	cmd : STRING := '?DST';
END_VAR
_deliverMessages := EFeedbackMsgSapphire488.DiodeSetTemperatureMsg;
_serialCom.Send(cmd);
END_METHOD

METHOD GetIdentifier
VAR_INPUT
END_VAR
VAR
	cmd : STRING := '?SV';
END_VAR
_deliverMessages := EFeedbackMsgSapphire488.IdMsg;
_serialCom.Send(cmd);
END_METHOD

(** Returns the status of the Interlock **)
METHOD PROTECTED GetInterlockStatus 
VAR_INPUT
END_VAR
VAR
	cmd : STRING := '?STA';
END_VAR
_deliverMessages := EFeedbackMsgSapphire488.InterlockStatusMsg;
_serialCom.Send(cmd);
END_METHOD

METHOD GetMeasuredTemperature 
VAR_INPUT
END_VAR
VAR
	cmd : STRING := '?DT';
END_VAR
_deliverMessages := EFeedbackMsgSapphire488.MeasuredTemperatureMsg;
_serialCom.Send(cmd);
END_METHOD

{attribute 'TcRpcEnable' := '1'}
(** Returns the timers of the laser and PSU:
		PSU Time=#######.#     Total time the system has been powered
		Laser Enabled Time=#######.#     Total time the diodes have been powered
		Laser OperationTime=#######.#    Total time the diodes have been powered >1 A  
**)
METHOD GetTimers : HoursStruct
VAR_INPUT
	Execute : BOOL;
END_VAR
VAR
	cmd : STRING := 'TIMERS?';
END_VAR
IF Execute THEN
	_logger.Information(_message.Reset().
								Append(_config.Name).
								Append(' - GetTimers').ToString());
	_serialCom.Send(cmd);
END_IF
END_METHOD

PROPERTY InitConfigSerialCom : BOOL
GET
InitConfigSerialCom := _initConfigSerialCom;
END_GET
SET
_initConfigSerialCom := InitConfigSerialCom;
END_SET
END_PROPERTY

METHOD InitDevice
VAR_INPUT
END_VAR
IF NOT _initDevice THEN	
	IF _pulseGenerator.Q THEN
		_pulseGenerator(IN := FALSE, PT := T#10MS);
			
		CASE _itemScheduler OF		
			0:	_logger.Information(_message.Reset().
								Append(_config.Name).
								Append(' - InitDevice').ToString());	

				_serialCom.Send('>=0'); // Echo off
				_itemScheduler := 1;				
		
			1:  _serialCom.Send('E=1'); // Set echo off
				_itemScheduler := 2;	
			
			2:  _serialCom.Send('T=1');  // Enable automatic servo regulation
				_itemScheduler := 3;	
    	
			3:	_raiseProperties:= TRUE;	
				_initDevice := TRUE;
				_itemScheduler := 0;
		END_CASE
	ELSE
	_pulseGenerator(IN := TRUE, PT := T#500MS);		
	END_IF
END_IF
END_METHOD

(** Returns the temperature of the laser head in degrees centigrade **)
METHOD LaserHeadReachedDiodeCurrentLimit 
VAR_INPUT
END_VAR
VAR
	cmd : STRING := '?MCR';
END_VAR
_deliverMessages := EFeedbackMsgSapphire488.LaserHeadReachedDiodeCurrentLimitMsg;
_serialCom.Send(cmd);
END_METHOD

METHOD MessageScheduler
VAR_INPUT
END_VAR
IF _pulseGenerator.Q THEN
	_pulseGenerator(IN := FALSE, PT := T#10MS);
		
	CASE _itemScheduler OF		
		0:	ReadPower();
			_itemScheduler := 1;				
	
		1:  GetBasePlateTemperature();
			_itemScheduler := 2;	
		
		2:  GetControllerTemperature();
			_itemScheduler := 3;		
			
		3:  GetDiodeSetTemperature();
			_itemScheduler := 4;
			
		4:  GetMeasuredTemperature();
			_itemScheduler := 5;
			
		5:  LaserHeadReachedDiodeCurrentLimit();
			_itemScheduler := 0;	
	END_CASE
ELSE
	_pulseGenerator(IN := TRUE, PT := T#500MS);		
END_IF
END_METHOD

{attribute 'TcRpcEnable' := '1'}
(** Disables the laser, regardless of the interlock status **)
METHOD PROTECTED PowerOff
VAR_INPUT
	Execute : BOOL;
END_VAR
VAR
	cmd : STRING := 'L=0';
END_VAR
IF Execute THEN	
	_powerOff := TRUE;	
	
	IF _execPulseGenerator.Q THEN
		_execPulseGenerator(IN := FALSE, PT := T#10MS);
			
		CASE _itemExecScheduler OF
			0: _logger.Information(_message.Reset().
								Append(_config.Name).
								Append(' - PowerOff').ToString());
				_serialCom.Send(cmd);
				_itemExecScheduler := 1;
			
			1:  GetInterlockStatus();
				_itemExecScheduler := 2;
				
			2:  _powerOff := FALSE;	
				_itemExecScheduler := 0;		
								
		END_CASE
	ELSE
		_execPulseGenerator(IN := TRUE, PT := T#500MS);	
	END_IF
END_IF
END_METHOD

{attribute 'TcRpcEnable' := '1'}
(* Enables the laser subject to Interlock and Enable Switch status *)
METHOD PROTECTED PowerOn
VAR_INPUT
	Execute : BOOL;
END_VAR
VAR
	cmd : STRING := 'L=1';
END_VAR
IF Execute THEN	
	_powerOn := TRUE;	

	IF _execPulseGenerator.Q THEN
		_execPulseGenerator(IN := FALSE, PT := T#10MS);
			
		CASE _itemExecScheduler OF
			0: _logger.Information(_message.Reset().
								Append(_config.Name).
								Append(' - PowerOn').ToString());
				_serialCom.Send(cmd);
				_itemExecScheduler := 1;
			
			1:  GetInterlockStatus();
				_itemExecScheduler := 2;
				
			2:  _powerOn := FALSE;	
				_itemExecScheduler := 0;		
								
		END_CASE
	ELSE
		_execPulseGenerator(IN := TRUE, PT := T#500MS);	
	END_IF
END_IF
END_METHOD

{attribute 'TcRpcEnable' := '1'}
METHOD RaisePropertiesChanged
VAR_INPUT
	Execute : BOOL;
END_VAR
IF Execute THEN
	_raiseProperties := TRUE;
	
	IF _pulseGenerator.Q THEN
		_pulseGenerator(IN := FALSE, PT := T#10MS);	

		CASE _itemRaisedProperties OF
			0:  InterlockStatusMsg := ' ';
				IdMsg := ' ';
				CustomMsg := ' ';
				
				_itemRaisedProperties := 10;
			
			10:  GetIdentifier();
				_itemRaisedProperties := 11;
				
			11:  GetInterlockStatus();
				_itemRaisedProperties := 12;
			
			12:  _logger.Information(_message.Reset().
								Append(_config.Name).
								Append(' - RaisePropertiesChanged').ToString());
				_raiseProperties := FALSE;				
				_itemRaisedProperties := 0;
			
		END_CASE
	ELSE
		_pulseGenerator(IN := TRUE, PT := T#500MS);	
	END_IF
END_IF
END_METHOD

(** Returns the power of the laser **)
METHOD PROTECTED ReadPower 
VAR_INPUT
END_VAR
VAR
	cmd : STRING := '?P';
END_VAR
_deliverMessages := EFeedbackMsgSapphire488.PowerMsg;	
_serialCom.Send(cmd);
END_METHOD

{attribute 'TcRpcEnable' := '1'}
(** This sets the output power of the laser 
For example, to set a power of 2800 mW, send the string POWER=2800, followed by striking the RETURN key
**)
METHOD PROTECTED SetPower 
VAR_INPUT
	Execute : BOOL;
	Power : LREAL;
END_VAR
VAR
	cmd : STRING := 'P=';
END_VAR
IF Execute THEN	
	_setPowerCmd := TRUE;	

	_setpoint := Power;
	
	IF _execPulseGenerator.Q THEN
		_execPulseGenerator(IN := FALSE, PT := T#10MS);
			
		CASE _itemExecScheduler OF
			0: _logger.Information(_message.Reset().
								Append(_config.Name).
								Append(' - SetPower : ').Append(TO_STRING(_setpoint)).ToString());
				_serialCom.Send(CONCAT(cmd, TO_STRING(_setpoint)));
				_itemExecScheduler := 1;
			
			1:  ReadPower();
				_itemExecScheduler := 2;
				
			2:  _setPowerCmd := FALSE;	
				_itemExecScheduler := 0;		
								
		END_CASE
	ELSE
		_execPulseGenerator(IN := TRUE, PT := T#500MS);	
	END_IF
END_IF
END_METHOD

END_FUNCTION_BLOCK

// ---- PMShared/Hardware/Devices/FiberSwitch/Leoni/EOLFiberSwitch.TcPOU
{attribute 'OPC.UA.DA' := '1'}
FUNCTION_BLOCK EOLFiberSwitch EXTENDS FiberSwitchBase
VAR_INPUT
END_VAR
VAR_OUTPUT
END_VAR
VAR
	{attribute 'OPC.UA.DA' := '0'}
	_config : EOLFiberSwitchConfig;
	{attribute 'OPC.UA.DA' := '0'}
	_coeAccess : CoeAccess;
	{attribute 'OPC.UA.DA' := '0'}
	_initConfigSerialCom : BOOL;
	{attribute 'OPC.UA.DA' := '0'}
	_serialCom  : SerialCom(Prefix :='', Suffix := Const.CARRIAGE_RETURN);
	{attribute 'OPC.UA.DA' := '0'}
	_refSerialCom : REFERENCE TO SerialCom(Prefix :='', Suffix := Const.CARRIAGE_RETURN) := _serialCom;	 
	{attribute 'OPC.UA.DA' := '0'}
	_isReceived : BOOL;
	
	{attribute 'OPC.UA.DA' := '0'}
	_deliverMessages : INT;
	
	IdMsg : STRING(255);
	CustomMsg : STRING(255);
	
	{region 'Commands'}
	
	{endregion}
	
	{attribute 'OPC.UA.DA' := '0'}
	_initDevice : BOOL;	
	 
	{attribute 'OPC.UA.DA' := '0'}
	_cmd : STRING;	
	{attribute 'OPC.UA.DA' := '0'}
	_itemScheduler : INT;		
	{attribute 'OPC.UA.DA' := '0'}
	_pulseGenerator : TON;	
			
	{attribute 'OPC.UA.DA' := '0'}
	message : STRING;
	{attribute 'OPC.UA.DA' := '0'}
	_length : INT;
		 
END_VAR


IF NOT InitConfigSerialCom THEN
	ConfigureSerialCom();
ELSE
	_refSerialCom(TxBuffer:= HardwareGlobalVariables.TxBufferFiberSwitch, 
		 	      RxBuffer:= HardwareGlobalVariables.RxBufferFiberSwitch);	
				  
	// Init device
	InitDevice(); 				  				 

	// Deliver messages
	IF _refSerialCom.IsReceived THEN
		_length := LEN(_refSerialCom.LastReceivedString);
		message := DELETE(_refSerialCom.LastReceivedString, 2, _length);
	
		CASE _deliverMessages OF			
			EFeedbackMsgEol.IdMsg :
				IdMsg := message;
			EFeedbackMsgEol.CustomMsg :
				CustomMsg := message;						
		END_CASE
		
		_deliverMessages := 0;
	END_IF					   	
END_IF

IF InitConfigSerialCom THEN	
	MessageScheduler();
END_IF

METHOD ConfigureSerialCom
VAR_INPUT
END_VAR
IF _coeAccess.CoeOperation.Ready THEN
	_logger.Information(_message.Reset().Append('Start configuration com serial').ToString());
END_IF;	

_coeAccess.CoeOperation.Start();
_coeAccess(SerialCommunication := _config.SerialCommunication);
	
IF _coeAccess.CoeOperation.Done THEN
	_coeAccess.SetDone();
	
	_Logger.Information(_message.Reset().
							Append('{').Append(TO_STRING(THIS^.Family)).Append('} : ').
							Append(' - Status : ').Append(TO_STRING(_coeAccess.Status)).ToString());	
	InitConfigSerialCom := TRUE;
END_IF
 
IF _coeAccess.CoeOperation.Error THEN	
	_coeAccess.SetError(0);
	
	_Logger.Error(_message.Reset().
							Append('{').Append(TO_STRING(THIS^.Family)).Append('} : ').
							Append(' - Status : ').Append(TO_STRING(_coeAccess.Status)).ToString());	
	InitConfigSerialCom := TRUE;
END_IF

THIS^.Status := _coeAccess.Status;
END_METHOD

{attribute 'TcRpcEnable' := '1'}
(** Response of the current switch position **)
METHOD PROTECTED CurrentPosition
VAR_INPUT
	Execute : BOOL;
END_VAR
VAR
	cmd : STRING := 'ch?';
END_VAR
IF Execute THEN
	_logger.Information(_message.Reset().
								Append(_config.Name).
								Append(' - CurrentPosition').ToString());
	_serialCom.Send(cmd);
END_IF
END_METHOD

METHOD FB_init : BOOL
VAR_INPUT
	bInitRetains : BOOL; // if TRUE, the retain variables are initialized (warm start / cold start)
	bInCopyCode : BOOL;  // if TRUE, the instance afterwards gets moved into the copy code (online change)
	Config : EOLFiberSwitchConfig;
END_VAR
IF Config.IsEnabled THEN
	_config := Config;
	
	SUPER^._fiberSwitchConfig.Name := Config.Name;
	SUPER^._fiberSwitchConfig.DeviceID := Config.DeviceID;
	SUPER^._fiberSwitchConfig.IsEnabled := Config.IsEnabled;
	SUPER^._fiberSwitchConfig.LogLevel := Config.LogLevel;
	
	SUPER^.Name := Config.Name;
	SUPER^.DeviceID := Config.DeviceID;	
	THIS^.Family := DeviceFamily.FiberSwitch;
		
	_Logger.Information(_message.Reset().Append('Init ').
							Append('{').Append(TO_STRING(THIS^.Family)).Append('} - ').
							Append('{').Append(TO_STRING(Config.Name)).Append('}').ToString());																													
END_IF
END_METHOD

{attribute 'TcRpcEnable' := '1'}
(** Response of the firmware version number **)
METHOD FirmwareVersion
VAR_INPUT
	Execute : BOOL;
END_VAR
VAR
	cmd : STRING := 'firmware?';
END_VAR
IF Execute THEN	
	_logger.Information(_message.Reset().
								Append(_config.Name).
								Append(' - FirmwareVersion').ToString());
	_serialCom.Send(cmd);
END_IF
END_METHOD

PROPERTY InitConfigSerialCom : BOOL
GET
InitConfigSerialCom := _initConfigSerialCom;
END_GET
SET
_initConfigSerialCom := InitConfigSerialCom;
END_SET
END_PROPERTY

METHOD InitDevice
VAR_INPUT
END_VAR
IF NOT _initDevice THEN	
	_logger.Information(_message.Reset().
								Append(_config.Name).
								Append(' - Init device').ToString());

	_initDevice := TRUE;	
END_IF
END_METHOD

METHOD MessageScheduler
VAR_INPUT
END_VAR
IF _pulseGenerator.Q THEN
	_pulseGenerator(IN := FALSE, PT := T#10MS);
		
	CASE _itemScheduler OF
		0:  
			_itemScheduler := 0;					
	END_CASE
ELSE
	_pulseGenerator(IN := TRUE, PT := T#50MS);	
END_IF
END_METHOD

{attribute 'TcRpcEnable' := '1'}
METHOD RaisePropertiesChanged
VAR_INPUT
	Execute : BOOL;
END_VAR
IF Execute THEN	
	IdMsg := ' ';
	CustomMsg := ' ';
END_IF
END_METHOD

{attribute 'TcRpcEnable' := '1'}
(** Sets the switch position **)
METHOD PROTECTED SetSwitchPosition
VAR_INPUT
	Execute : BOOL;
	Position : UINT;
END_VAR
VAR
	cmd : STRING := 'ch';
END_VAR
IF Execute THEN	
	_logger.Information(_message.Reset().
								Append(_config.Name).
								Append(' - SetSwitchPosition : ').Append(TO_STRING(Position)).ToString());
	_serialCom.Send(CONCAT(cmd, TO_STRING(Position)));
	
END_IF
END_METHOD

{attribute 'TcRpcEnable' := '1'}
(** Response of the switch type **)
METHOD SwitchType
VAR_INPUT
	Execute : BOOL;
END_VAR
VAR
	cmd : STRING := 'type?';
END_VAR
IF Execute THEN	
	_logger.Information(_message.Reset().
								Append(_config.Name).
								Append(' - SwitchType').ToString());
	_serialCom.Send(cmd);
END_IF
END_METHOD

END_FUNCTION_BLOCK

// ---- PMShared/Hardware/Devices/FiberSwitch/FiberSwitchBase.TcPOU
FUNCTION_BLOCK ABSTRACT FiberSwitchBase EXTENDS TExecution IMPLEMENTS IDevice
VAR_INPUT
END_VAR
VAR_OUTPUT
END_VAR
VAR
	{attribute 'OPC.UA.DA' := '0'}
	_name : STRING;
	{attribute 'OPC.UA.DA' := '0'}
	_deviceID : STRING;					
	{attribute 'OPC.UA.DA' := '0'}
	_family : DeviceFamily;	
	{attribute 'OPC.UA.DA' := '0'}	
	_logger : Logger;
	{attribute 'OPC.UA.DA' := '0'}
	_message : StringBuilder;
	{attribute 'OPC.UA.DA' := '0'}
	_fiberSwitchConfig : DeviceConfiguration;
END_VAR

METHOD PROTECTED ABSTRACT CurrentPosition
VAR_INPUT
	Execute : BOOL;
END_VAR
END_METHOD

PROPERTY DeviceID : STRING
GET
DeviceID := _deviceID;
END_GET
SET
_deviceID := DeviceID;
END_SET
END_PROPERTY

PROPERTY Family : DeviceFamily
GET
Family := _family;
END_GET
SET
_family := Family;
END_SET
END_PROPERTY

PROPERTY Name : STRING
GET
Name := _name;
END_GET
SET
_name := Name;
END_SET
END_PROPERTY

METHOD PROTECTED ABSTRACT SetSwitchPosition
VAR_INPUT
	Execute : BOOL;
	Position : UINT;
END_VAR
END_METHOD

END_FUNCTION_BLOCK

// ---- PMShared/Hardware/Devices/OpticalPowermeters/Thorlabs/PM101/PM101OpticalPowermeterHs.TcPOU
{attribute 'OPC.UA.DA' := '1'}
FUNCTION_BLOCK PM101OpticalPowermeterHs EXTENDS PM101OpticalPowermeter
VAR_INPUT
END_VAR
VAR_OUTPUT
END_VAR
VAR
	{attribute 'OPC.UA.DA' := '0'}
	_config : PM101OpticalPowermeterConfig;
	{attribute 'OPC.UA.DA' := '0'}
	_polarisationConfig : PolarisationConfig;
	{attribute 'OPC.UA.DA' := '0'}
	_responsivityConfig : ResponsivityConfig;
	{attribute 'OPC.UA.DA' := '0'}
	_rFactorSettings : RFactorSettings;
	{attribute 'OPC.UA.DA' := '0'}
	_coeAccess : CoeAccess;
	{attribute 'OPC.UA.DA' := '0'}
	_initConfigSerialCom : BOOL;
	{attribute 'OPC.UA.DA' := '0'}	
	_serialCom  : SerialCom(Prefix :='', Suffix := Const.LINE_FEED);
	{attribute 'OPC.UA.DA' := '0'}
	_refSerialCom : REFERENCE TO SerialCom(Prefix :='', Suffix := Const.LINE_FEEL) := _serialCom;	
	
	{attribute 'OPC.UA.DA' := '0'}
	_pulseGeneratorInit : TON;	
	{attribute 'OPC.UA.DA' := '0'}
	_itemInit : INT;
END_VAR

IF _config.IsSimulated THEN
	SUPER^(Conf := _config, PolarisationConfig := _polarisationConfig, RFactorSettings := _rfactorSettings, ResponsivityConfig := _responsivityConfig, SerialCom := _serialCom, RefSerialCom := _refSerialCom);
ELSE
	IF NOT InitConfigSerialCom THEN
		ConfigureSerialCom();
	ELSIF THIS^.Status = TExecutionState.Ready THEN
		IF _refSerialCom.ErrorReceiveId = COMERROR_NOERROR THEN
			_refSerialCom(TxBuffer:= HardwareGlobalVariables.TxBufferOpticalPowermeterHs, 
						  RxBuffer:= HardwareGlobalVariables.RxBufferOpticalPowermeterHs);
		END_IF						  			
					
		SUPER^(Conf := _config, PolarisationConfig := _polarisationConfig, RFactorSettings := _rfactorSettings, ResponsivityConfig := _responsivityConfig, SerialCom := _serialCom, RefSerialCom := _refSerialCom);

		// Init device
		InitDevice(); 			
	END_IF
END_IF

METHOD ConfigureSerialCom
VAR_INPUT
END_VAR
IF _coeAccess.CoeOperation.Ready THEN
	_logger.Information(_message.Reset().Append('Start configuration com serial').ToString());
END_IF;	

_coeAccess.CoeOperation.Start();
_coeAccess(SerialCommunication := _config.SerialCommunication);
	
IF _coeAccess.CoeOperation.Done THEN
	_coeAccess.SetDone();
	
	_Logger.Information(_message.Reset().
							Append('{').Append(TO_STRING(THIS^.Family)).Append('} : ').
							Append(' - Status : ').Append(TO_STRING(_coeAccess.Status)).ToString());
	InitConfigSerialCom := TRUE;
END_IF
 
IF _coeAccess.CoeOperation.Error THEN	
	_coeAccess.SetError(0);
	
	_Logger.Error(_message.Reset().
							Append('{').Append(TO_STRING(THIS^.Family)).Append('} : ').
							Append(' - Status : ').Append(TO_STRING(_coeAccess.Status)).ToString());
	InitConfigSerialCom := TRUE;
END_IF

THIS^.Status := _coeAccess.Status;
State := _coeAccess.Status;
END_METHOD

METHOD FB_init : BOOL
VAR_INPUT
	bInitRetains : BOOL; // if TRUE, the retain variables are initialized (warm start / cold start)
	bInCopyCode : BOOL;  // if TRUE, the instance afterwards gets moved into the copy code (online change)
	Config : PM101OpticalPowermeterConfig;
	PolarisationConfig : PolarisationConfig;
	RFactorSettings : RFactorSettings;
	ResponsivityConfig : ResponsivityConfig;
END_VAR
IF Config.IsEnabled THEN
	_config := Config;
	_polarisationConfig := PolarisationConfig;
	_rFactorSettings := RFactorSettings;
	_responsivityConfig := ResponsivityConfig;
	
	SUPER^._opticalPowermeterConfig.Name := Config.Name;
	SUPER^._opticalPowermeterConfig.DeviceID := Config.DeviceID;
	SUPER^._opticalPowermeterConfig.IsEnabled := Config.IsEnabled;
	SUPER^._opticalPowermeterConfig.LogLevel := Config.LogLevel;
	
	SUPER^.Name := Config.Name;
	SUPER^.DeviceID := Config.DeviceID;	
	THIS^.Family := DeviceFamily.OpticalPowermeter;
		
	_Logger.Information(_message.Reset().Append('Init ').
							Append('{').Append(TO_STRING(THIS^.Family)).Append('} - ').
							Append('{').Append(TO_STRING(Config.Name)).Append('}').ToString());																													
END_IF
END_METHOD

PROPERTY InitConfigSerialCom : BOOL
GET
InitConfigSerialCom := _initConfigSerialCom;
END_GET
SET
_initConfigSerialCom := InitConfigSerialCom;
END_SET
END_PROPERTY

METHOD InitDevice 
VAR_INPUT	
END_VAR
IF NOT _initDevice THEN	
	CASE _itemInit OF
		0:  _logger.Information(_message.Reset().Append(_config.Name).Append(' - InitDevice').ToString());
			_itemInit := 1;
		
		1:  SUPER^._rangeAuto := TRUE;
			SUPER^._cmdRange := 'TRUE';
			_itemInit := 2;			
			
		2:  SUPER^._setSensorAttenuation := TRUE;
			SUPER^._cmdSensorAttenuation := _config.Sensor.Attenuation;
			_itemInit := 3;
			
		3:  IF _config.Sensor.Name = Const.POWERMETER_SENSOR_NAME_S150C THEN
				_logger.Error(_message.Reset().Append(_config.Name).Append(' - Sensor name: ').Append(_config.Sensor.Name).ToString());
				_itemInit := 10;
			ELSIF _config.Sensor.Name = Const.POWERMETER_SENSOR_NAME_TAP_COUPLER THEN
				_logger.Error(_message.Reset().Append(_config.Name).Append(' - Sensor name: ').Append(_config.Sensor.Name).ToString());
				_itemInit := 20;
			ELSE
				_logger.Error(_message.Reset().Append(_config.Name).Append(' - NAME OF FAILED SENSOR').ToString());
		    END_IF
			
		10:  SUPER^._setWavelength := TRUE;
			 SUPER^._cmdWavelength := _config.Sensor.Wavelength;
			 _itemInit := 50;		
		
		20:  GetResponsivity();
			 _itemInit := 21;
			
		21:	 _pulseGeneratorInit(IN := TRUE, PT := T#3000MS);
			 IF _pulseGeneratorInit.Q THEN
				_pulseGeneratorInit(IN := FALSE);				
			 	_itemInit := 22;
			 END_IF
		
		22:	 IF ResponsivityMsg = LREAL_TO_STRING(_responsivityConfig.Responsivity_mA_W) THEN
			 	_logger.Information(_message.Reset().Append(_config.Name).Append(' - Responsivity already defined').ToString());
			 	_itemInit := 50;
			 ELSE				 
				_itemInit := 23;
			 END_IF	
			 
		23:  _logger.Information(_message.Reset().
							Append(_config.Name).
							Append(' - Init responsivity: ').
							Append(LREAL_TO_STRING(_responsivityConfig.Responsivity_mA_W)).ToString());
			
			SUPER^._setpoint := _responsivityConfig.Responsivity_ma_W;
			SUPER^._setResponsivity := TRUE;
			
			_itemInit := 50;

		50: _logger.Information(_message.Reset().
							Append(_config.Name).
							Append(' - InitDevice done').ToString());				
			_initDevice	:= TRUE;
	END_CASE			
END_IF
END_METHOD

END_FUNCTION_BLOCK

// ---- PMShared/Hardware/Devices/OpticalPowermeters/Thorlabs/PM101OpticalPowermeter.TcPOU
{attribute 'OPC.UA.DA' := '1'}
FUNCTION_BLOCK PM101OpticalPowermeter EXTENDS OpticalPowermeterBase
VAR_INPUT
	{attribute 'OPC.UA.DA' := '0'}
	Conf : PM101OpticalPowermeterConfig;
	{attribute 'OPC.UA.DA' := '0'}
	PolarisationConfig : PolarisationConfig;
	{attribute 'OPC.UA.DA' := '0'}
	RFactorSettings : RFactorSettings;
	{attribute 'OPC.UA.DA' := '0'}
	ResponsivityConfig : ResponsivityConfig;	
	{attribute 'OPC.UA.DA' := '0'}	
	SerialCom  : SerialCom(Prefix :='', Suffix := Const.LINE_FEED); 
	{attribute 'OPC.UA.DA' := '0'}
	RefSerialCom : REFERENCE TO SerialCom(Prefix :='', Suffix := Const.LINE_FEED) := SerialCom; 
	{attribute 'OPC.UA.DA' := '0'}
	PolarResult : EPolar;	 
END_VAR
VAR_OUTPUT
END_VAR
VAR
	{attribute 'OPC.UA.DA' := '0'}
	IoControlPM101 : IoControlPM101;	

	{attribute 'OPC.UA.DA' := '0'}
	_deliverMessages : INT;
		
	PowerMsg : STRING(255);
	CurrentMsg : STRING(255);		
	IdentifierMsg : STRING(255);
	ResponsivityMsg : STRING(255) := 'Undefined';
	DarkOffsetMsg : STRING(255);
	DarkAdjustStateMsg : STRING(255);
	CustomMsg : STRING(255);	
	SensorTypeMsg : STRING(255);			
	WavelengthMsg : STRING(255);				
	(* Not necessary *)
	BeamDiameterMsg : STRING(255);
	SensorAttenuationMsg : STRING(255);			
	MaxPowerMsg : STRING(255);
	MinPowerMsg : STRING(255);
	WavelengthRangeMsg : STRING(255);	
	CalibMsg : STRING(255);
	
	
	{attribute 'OPC.UA.DA' := '0'}
	_flow : STRING;
	{attribute 'OPC.UA.DA' := '0'}
	_powerRawAbs : LREAL;
	{attribute 'OPC.UA.DA' := '0'}
	_powerCal_mW : LREAL;	
	{attribute 'OPC.UA.DA' := '0'}
	_powerRaw_mW : LREAL;
	{attribute 'OPC.UA.DA' := '0'}
	_current_mA : LREAL;
	{attribute 'OPC.UA.DA' := '0'}
	_darkAdjustState : STRING(255);
	{attribute 'OPC.UA.DA' := '0'}	
	_darkOffset_mW : LREAL;
	{attribute 'OPC.UA.DA' := '0'}	
	_responsivity_mW_mA : LREAL;
	{attribute 'OPC.UA.DA' := '0'}
	_rfactor : LREAL := -1;
	
	{region 'Commands'}
	
	{attribute 'OPC.UA.DA' := '0'}		 
	_abortCmd : BOOL;
	{attribute 'OPC.UA.DA' := '0'}	
	_customCmd : BOOL;	
	{attribute 'OPC.UA.DA' := '0'}
	_setBeamDiameter : BOOL;	
	{attribute 'OPC.UA.DA' := '0'}
	_setWavelength : BOOL;	
	{attribute 'OPC.UA.DA' := '0'}
	 _rangeAuto : BOOL;
	{attribute 'OPC.UA.DA' := '0'}	  
	_setSensorAttenuation : BOOL;
	{attribute 'OPC.UA.DA' := '0'} 		
	_setSensorType : BOOL;	 	
	{attribute 'OPC.UA.DA' := '0'}			  		   
	_raiseProperties : BOOL;
	{attribute 'OPC.UA.DA' := '0'}
	_rangeVariation : BOOL;
	{attribute 'OPC.UA.DA' := '0'}
	_startDarkAdjust : BOOL;	 
	{attribute 'OPC.UA.DA' := '0'}
	_cancelDarkAdjust : BOOL;	
	{attribute 'OPC.UA.DA' := '0'}
	_setResponsivity : BOOL; 
	{endregion}
	
	{attribute 'OPC.UA.DA' := '0'}
	_initDevice : BOOL;	
	{attribute 'OPC.UA.DA' := '0'}
	_monitoringMessages : BOOL;	
	 
	{attribute 'OPC.UA.DA' := '0'}
	_cmd : STRING;
	{attribute 'OPC.UA.DA' := '0'}
	_cmdRange : STRING;
	{attribute 'OPC.UA.DA' := '0'}
	_cmdRangesVariation : STRING;
	{attribute 'OPC.UA.DA' := '0'}
	_cmdBeamDiameter : UINT;
	{attribute 'OPC.UA.DA' := '0'}
	_cmdWavelength : UINT;	
	{attribute 'OPC.UA.DA' := '0'}
	_cmdSensorAttenuation : UINT;	
	{attribute 'OPC.UA.DA' := '0'}
	_cmdSensorType : STRING;
	{attribute 'OPC.UA.DA' := '0'}
	_setpoint : LREAL := 0;
	{attribute 'OPC.UA.DA' := '0'}
	_itemScheduler : INT;
	{attribute 'OPC.UA.DA' := '0'}
	_itemExecScheduler : INT;
	{attribute 'OPC.UA.DA' := '0'}
	_itemRaisedProperties : INT;	
	{attribute 'OPC.UA.DA' := '0'}
	_itemSchedulerResponsivity : INT;	
	{attribute 'OPC.UA.DA' := '0'}
	_pulseGenerator : TON;
	{attribute 'OPC.UA.DA' := '0'}
	_pulseGeneratorMsg : TON;
	{attribute 'OPC.UA.DA' := '0'}
	_pulseGeneratorCmd : TON;
	{attribute 'OPC.UA.DA' := '0'}
	_execPulseGenerator : TON;	
	{attribute 'OPC.UA.DA' := '0'}
	_pulseGeneratorCustom : TON;		
	
	{attribute 'OPC.UA.DA' := '0'}
	message : STRING;
	{attribute 'OPC.UA.DA' := '0'}
	_length : INT;
		
	{attribute 'OPC.UA.DA' := '0'}
	_illumFlow : STRING := ' ';
	{attribute 'OPC.UA.DA' := '0'}
	_delimeter : STRING := ';';
	{attribute 'OPC.UA.DA' := '0'}
	_firstConcat : STRING;
	{attribute 'OPC.UA.DA' := '0'}
	_secondConcat : STRING;
	{attribute 'OPC.UA.DA' := '0'}
	_thirdConcat : STRING;
	{attribute 'OPC.UA.DA' := '0'}
	_fourthConcat : STRING;
	{attribute 'OPC.UA.DA' := '0'}
	_fifthConcat : STRING;
	{attribute 'OPC.UA.DA' := '0'}
	_sixthConcat : STRING;
	{attribute 'OPC.UA.DA' := '0'}
	_seventhConcat : STRING;
END_VAR

IF _illumFlow = ' ' THEN	
	IF (Conf.DeviceID = TO_STRING(EPowerIlluminationFlow.HS)) THEN
		_flow := TO_STRING(EPowerIlluminationFlow.HS);
	ELSE
		_flow := TO_STRING(EPowerIlluminationFlow.HT);
	END_IF	
		
	_illumFlow := CONCAT(_flow, _delimeter);
END_IF		


// Deliver messages
IF RefSerialCom.IsReceived OR Conf.IsSimulated THEN					
	IF NOT Conf.IsSimulated THEN
		_length := LEN(RefSerialCom.LastReceivedString);
		message := DELETE(RefSerialCom.LastReceivedString, 2, _length);
	END_IF
		
	IF _monitoringMessages THEN
		CASE _deliverMessages OF			
			EFeedbackMsgPM101.PowerMsg :
				
				IF PolarResult = EPolar.S_Polar THEN
					_rfactor := RFactorSettings.RFactor_S;
				ELSIF PolarResult = EPolar.P_Polar THEN
					_rfactor := RFactorSettings.RFactor_P;
				END_IF			
				
				_powerRawAbs := ABS(STRING_TO_LREAL(message));
				IF  _powerRawAbs > 0 THEN						
					_powerRaw_mW := _powerRawAbs * 1000;
					_powerCal_mW := _powerRawAbs * 1000 / _rfactor;
					
					_firstConcat := CONCAT(_illumFlow, TO_STRING(_powerRaw_mW));	
					_secondConcat := CONCAT(_firstConcat, _delimeter);	
					_thirdConcat := CONCAT(_secondConcat, TO_STRING(_powerCal_mW));
					_fourthConcat := CONCAT(_thirdConcat, _delimeter);
					
					PowerMsg :=  CONCAT(_fourthConcat, TO_STRING(_rfactor));
				END_IF
			EFeedbackMsgPM101.CurrentMsg :				
				_current_mA := STRING_TO_LREAL(message) * 1000;		
				CurrentMsg := CONCAT(_illumFlow, TO_STRING(_current_mA));	
		END_CASE
	ELSE
		CASE _deliverMessages OF
			EFeedbackMsgPM101.IdentifierMsg :				   		
				IdentifierMsg := CONCAT(_illumFlow, message);
				_logger.Information(_message.Reset().Append('IdentifierMsg: ').Append(IdentifierMsg).ToString());													
			EFeedbackMsgPM101.ResponsivityMsg :			
				_responsivity_mW_mA := (STRING_TO_LREAL(message) * 1E3);		
				ResponsivityMsg := CONCAT(_illumFlow, TO_STRING(_responsivity_mW_mA));	
				_logger.Information(_message.Reset().Append('ResponsivityMsg: ').Append(ResponsivityMsg).ToString());						
				message := ' ';	
				
			EFeedbackMsgPM101.DarkOffsetMsg :						
				_darkOffset_mW := (STRING_TO_LREAL(message) * 1E12); 			
				DarkOffsetMsg := CONCAT(_illumFlow, TO_STRING(_darkOffset_mW));	
				_logger.Information(_message.Reset().Append('DarkOffsetMsg: ').Append(DarkOffsetMsg).ToString());	
			EFeedbackMsgPM101.DarkAdjustStateMsg :				
				DarkAdjustStateMsg := CONCAT(_illumFlow, message);			
				_logger.Information(_message.Reset().Append('DarkAdjustStateMsg: ').Append(DarkAdjustStateMsg).ToString());	
									
			EFeedbackMsgPM101.CustomMsg :		    	
				CustomMsg := CONCAT(_illumFlow, message);	
				_logger.Information(_message.Reset().Append('CustomMsg: ').Append(CustomMsg).ToString());
				
				
			EFeedbackMsgPM101.SensorTypeMsg :				
				SensorTypeMsg := CONCAT(_illumFlow, message);					
			EFeedbackMsgPM101.WavelengthMsg :			
				WavelengthMsg := CONCAT(_illumFlow, message);
			EFeedbackMsgPM101.BeamDiameterMsg :			
				BeamDiameterMsg := CONCAT(_illumFlow, message);			
			EFeedbackMsgPM101.SensorAttenuationMsg :			
				SensorAttenuationMsg := CONCAT(_illumFlow, message);	
			EFeedbackMsgPM101.WavelengthRangeMsg :
				WavelengthRangeMsg := CONCAT(_illumFlow, message);	
			EFeedbackMsgPM101.MaxPowerMsg :
				MaxPowerMsg := CONCAT(_illumFlow, message);
			EFeedbackMsgPM101.MinPowerMsg :
				MinPowerMsg := CONCAT(_illumFlow, message);	
		END_CASE
	END_IF							
	
ELSE
	CASE _deliverMessages OF
		EFeedbackMsgPM101.CalibMsg :				
			_fifthConcat := CONCAT(_illumFlow, LREAL_TO_FMTSTR(RFactorSettings.RFactor_S, 10, TRUE));	
			_sixthConcat := CONCAT(_fifthConcat, _delimeter);
			_seventhConcat := CONCAT(_sixthConcat, LREAL_TO_FMTSTR(RFactorSettings.RFactor_P, 10, TRUE));	
		
			CalibMsg := _seventhConcat;
	END_CASE	
END_IF

// Commands
EnableAutoRange(_rangeAuto, STRING_TO_BOOL(_cmdRange));
RangesVariation(_rangeVariation, _cmdRangesVariation);
StartDarkAdjust(_startDarkAdjust);
CancelDarkAdjust(_cancelDarkAdjust);
Abort(_abortCmd);
RaisePropertiesChanged(_raiseProperties);
CustomCommand(_customCmd, _cmd);

// For init sensor
SetResponsivity(_setResponsivity, _setpoint);
SetBeamDiameter(_setBeamDiameter, _cmdBeamDiameter);
SetWavelength(_setWavelength, _cmdWavelength);
SetSensorAttenuation(_setSensorAttenuation, _cmdSensorAttenuation);
SetSensorType(_setSensorType, _cmdSensorType);

// Monitoring some values 
IF _monitoringMessages THEN
	MessageScheduler();
END_IF

(*
IF (NOT _setBeamDiameter AND NOT _setWavelength AND NOT _rangeAuto AND NOT _setSensorAttenuation
    AND NOT _setSensorType AND NOT _setResponsivity AND NOT _customCmd AND NOT _raiseProperties 
	AND NOT _rangeVariation AND NOT _startDarkAdjust AND NOT _cancelDarkAdjust AND NOT _abortCmd) THEN
	MessageScheduler();
END_IF	
*)

METHOD Abort : BOOL;
VAR_INPUT
	Execute : BOOL;
END_VAR
VAR_OUTPUT
	Stop : BOOL;
END_VAR
VAR
	cmd : STRING := 'ABORt';
END_VAR
IF Execute THEN
	_logger.Information(_message.Reset().
								Append(Conf.Name).
								Append(' - Abort command').ToString());																
	SerialCom.Send(Cmd);	
	_abortCmd := FALSE;
	
	//ABORT := TRUE;		 
END_IF
END_METHOD

{attribute 'TcRpcEnable' := '1'}
METHOD CancelDarkAdjust
VAR_INPUT
	Execute : BOOL;
END_VAR
VAR	
	cmd : STRING := 'Sense:CORRection:COLLect:ZERO:ABORt';	
END_VAR
IF Execute THEN
	_logger.Information(_message.Reset().
								Append(Conf.Name).
								Append(' - Cancel dark adjust').ToString());
	
	//Abort(_abortCmd);
	SerialCom.Send(cmd);
	_cancelDarkAdjust := FALSE;
END_IF
END_METHOD

{attribute 'TcRpcEnable' := '1'}
(** Custom command **)
METHOD CustomCommand
VAR_INPUT
	Execute : BOOL;
	Cmd : STRING;
END_VAR
IF Execute THEN
	_logger.Information(_message.Reset().
								Append(Conf.Name).
								Append(' - Custom command:').
								Append(Cmd).ToString());
	
	_deliverMessages := EFeedbackMsgPM101.CustomMsg;																								
	SerialCom.Send(Cmd);	
	_customCmd := FALSE;
END_IF

(*
IF Execute THEN
	IF _pulseGeneratorCustom.Q THEN
		_pulseGeneratorCustom(IN := FALSE);									
		_customCmd := FALSE;
	ELSE	
		_pulseGeneratorCustom(IN := Execute, PT := T#100MS);										
	END_IF	
END_IF	
*)
END_METHOD

{attribute 'TcRpcEnable' := '1'}
(** Switches the auto-ranging function on and off **)
METHOD EnableAutoRange
VAR_INPUT
	Execute : BOOL;
	Activate : BOOL;
END_VAR
VAR
	cmd : STRING := 'Sense:Power:Dc:Range:AUTO ';
	autorRange : STRING;
END_VAR
IF Execute THEN
	_logger.Information(_message.Reset().
								Append(Conf.Name).
								Append(' - Switches the auto-ranging: ').
								Append(TO_STRING(Activate)).ToString());
	
	IF Activate THEN
		autorRange := 'Sense:Power:Dc:Range:AUTO ON';
	ELSE
		autorRange := 'Sense:Power:Dc:Range:AUTO OFF';
	END_IF
					
	SerialCom.Send(CONCAT(cmd, TO_STRING(Activate)));	
	_rangeAuto := FALSE;
END_IF
END_METHOD

METHOD GetBeamDiameter
VAR_INPUT
END_VAR
VAR	
	cmd : STRING := 'Sense:Correction:beamdiameter? ';	
END_VAR
_logger.Information(_message.Reset().Append('GetBeamDiameter').ToString());
_deliverMessages := EFeedbackMsgPM101.BeamDiameterMsg;

IF NOT Conf.IsSimulated THEN
	SerialCom.Send(cmd);
ELSE
	message := '5';
END_IF
END_METHOD

(** Read the unit’s identification string **)
METHOD GetCalibConfig
VAR_INPUT
END_VAR
VAR
END_VAR
_deliverMessages := EFeedbackMsgPM101.CalibMsg;
END_METHOD

METHOD GetDarkAdjustState
VAR_INPUT
END_VAR
VAR	
	cmd : STRING := 'Sense:Correction:COLLect:ZERO:STATe?';	
END_VAR
_deliverMessages := EFeedbackMsgPM101.DarkAdjustStateMsg;					

IF NOT Conf.IsSimulated THEN
	SerialCom.Send(cmd);
ELSE
	message := 'Simu_ok';
END_IF
END_METHOD

METHOD GetDarkOffset
VAR_INPUT
END_VAR
VAR	
	cmd : STRING := 'Sense:CORRection:COLLect:ZERO:MAGNitude?';	
END_VAR
_deliverMessages := EFeedbackMsgPM101.DarkOffsetMsg;
SerialCom.Send(cmd);
END_METHOD

(** Read the unit’s identification string **)
METHOD GetIdentifier
VAR_INPUT
END_VAR
VAR
	cmd : STRING := 'System:Sensor:IDN?';
END_VAR
_deliverMessages := EFeedbackMsgPM101.IdentifierMsg;
SerialCom.Send(cmd);
END_METHOD

(** Get max measure power **)
METHOD GetMaxPower
VAR_INPUT
END_VAR
VAR	
	cmd : STRING := 'Measure:Scalar:POWer? MAXimum';	
END_VAR
_deliverMessages := EFeedbackMsgPM101.MaxPowerMsg;					
SerialCom.Send(cmd);
END_METHOD

(** Get in measure power **)
METHOD GetMinPower
VAR_INPUT
END_VAR
VAR	
	cmd : STRING := 'Measure:Scalar:POWer? MINimum';	
END_VAR
_deliverMessages := EFeedbackMsgPM101.MinPowerMsg;	
SerialCom.Send(cmd);
END_METHOD

METHOD GetResponsivity
VAR_INPUT
END_VAR
VAR	
	cmd : STRING := 'Sense:Correction:power:pdiode:response?';	
END_VAR
_deliverMessages := EFeedbackMsgPM101.ResponsivityMsg;

IF Conf.IsSimulated THEN
	message := LREAL_TO_STRING(0.05);
ELSE
	SerialCom.Send(cmd);	
END_IF
END_METHOD

(** Get the beam diameter in mm **)
METHOD GetSensorAttenuation
VAR_INPUT
END_VAR
VAR	
	cmd : STRING := 'Sense:Correction:BEAMdiameter? ';	
END_VAR
//_logger.Information(_message.Reset().Append('GetSensorAttenuation').ToString());
_deliverMessages := EFeedbackMsgPM101.SensorAttenuationMsg;

IF NOT Conf.IsSimulated THEN
	SerialCom.Send(cmd);
ELSE
	message := INT_TO_STRING(2);
END_IF
END_METHOD

METHOD GetSensorType
VAR_INPUT
END_VAR
VAR	
	cmd : STRING := 'Input:Adapter:TYPE?';	
END_VAR
//_logger.Information(_message.Reset().Append('GetSensorType').ToString());
_deliverMessages := EFeedbackMsgPM101.SensorTypeMsg;

IF Conf.IsSimulated THEN
	message := 'SIMU_PHOTODIODE';	
ELSE
	SerialCom.Send(cmd);
END_IF



(*IF _pulseGeneratorCmd.Q THEN
	_pulseGeneratorCmd(IN := FALSE, PT := T#10MS);	
								
	SerialCom.Send(cmd);
ELSE
	_deliverMessages := EFeedbackMsgPM101.SensorTypeMsg;
	_pulseGeneratorCmd(IN := TRUE, PT := T#100MS);										
END_IF	*)
END_METHOD

(** Get wavelength **)
METHOD GetWavelength
VAR_INPUT
END_VAR
VAR	
	cmd : STRING := 'Sense:CORR:WAVE?';	
END_VAR
_deliverMessages := EFeedbackMsgPM101.WavelengthMsg;

IF Conf.IsSimulated THEN
	message := INT_TO_STRING(473);
ELSE	
	SerialCom.Send(cmd);
END_IF	


(*IF _pulseGeneratorCmd.Q THEN
	_pulseGeneratorCmd(IN := FALSE, PT := T#10MS);	
								
	SerialCom.Send(cmd);
ELSE
	_deliverMessages := EFeedbackMsgPM101.WavelengthMsg;
	_pulseGeneratorCmd(IN := TRUE, PT := T#100MS);										
END_IF*)
END_METHOD

(** Get wavelength range **)
METHOD GetWavelengthRange
VAR_INPUT
END_VAR
VAR	
	cmd : STRING := 'Sense:Power:Dc:Range:UPPer? MINimum ';	
END_VAR
_deliverMessages := EFeedbackMsgPM101.WavelengthRangeMsg;
SerialCom.Send(cmd);
END_METHOD

METHOD MessageScheduler
VAR_INPUT
END_VAR
IF _pulseGenerator.Q THEN
	_pulseGenerator(IN := FALSE, PT := T#10MS);
		
	CASE _itemScheduler OF		   
		0:	ReadPower();	
			_itemScheduler := 1;
			
		1: ReadCurrent();			
		   _itemScheduler := 0;
	END_CASE
ELSE
	_pulseGenerator(IN := TRUE, PT := T#50MS);	
END_IF


(*CASE _itemScheduler OF
	0:  _pulseGeneratorMsg(IN := TRUE, PT := T#10MS); // 50MS + 10MS de temps de cycle = 60 MS 
		IF _pulseGeneratorMsg.Q THEN
			_pulseGeneratorMsg(IN := FALSE);			
			
			ReadPower();			
			_itemScheduler := 1;
		END_IF 

	1:  _pulseGeneratorMsg(IN := TRUE, PT := T#100MS); // 50MS + 10MS de temps de cycle = 60 MS 
		IF _pulseGeneratorMsg.Q THEN
			_pulseGeneratorMsg(IN := FALSE);			
			
			ReadCurrent();			
			_itemScheduler := 0;
		END_IF  												
END_CASE
*)
END_METHOD

{attribute 'TcRpcEnable' := '1'}
METHOD RaisePropertiesChanged
VAR_INPUT
	Execute : BOOL;
END_VAR
IF Execute THEN	
	_monitoringMessages := FALSE;
	_raiseProperties := TRUE;
	
	CASE _itemRaisedProperties OF		
		0: IdentifierMsg := ' ';
		   ResponsivityMsg := ' ';
		   CustomMsg := ' ';
		   WavelengthMsg := ' ';
		   BeamDiameterMsg := ' ';
		   WavelengthRangeMsg := ' ';				   	 
  		   SensorTypeMsg := ' ';
		   CalibMsg := ' ';
		   _itemRaisedProperties := 10;																																								
			
		10: GetCalibConfig();
			_itemRaisedProperties := 50;	

		11:  _logger.Information(_message.Reset().Append(Conf.Name).Append(' RaisedProperties- Get responsivity').ToString());
			GetResponsivity();
			_itemRaisedProperties := 12;
			
		12: IF message = ' ' THEN
			  _itemRaisedProperties := 50;
			END_IF	
			
		(* Not necessary *)
		(*
		10: GetIdentifier();
			_itemRaisedProperties := 11;
			
		11: GetSensorType();
			_itemRaisedProperties := 12;
		
		12: GetWavelength();
			_itemRaisedProperties := 13;	
    
		12: GetBeamDiameter();
			_itemRaisedProperties := 16;
	
		13: GetWavelengthRange();
			_itemRaisedProperties := 16;
	
		14:  GetMaxPower();
			_itemRaisedProperties := 15;
			
		15: GetMinPower();
			_itemRaisedProperties := 16;
			
		17: GetSensorAttenuation();
			_itemRaisedProperties := 19;*)
			
		50: 
			_logger.Information(_message.Reset().
							    Append(Conf.Name).
							    Append(' - RaisePropertiesChanged').ToString());
			_raiseProperties := FALSE;				
			_itemRaisedProperties := 0;
	
			_monitoringMessages := TRUE;								
	END_CASE
END_IF

(*IF Execute THEN	
	_raiseProperties := TRUE;
	
	IF _pulseGenerator.Q THEN
		_pulseGenerator(IN := FALSE);
	
		CASE _itemRaisedProperties OF		
			0: IdentifierMsg := ' ';
			   ResponsivityMsg := ' ';
			   CustomMsg := ' ';
			   WavelengthMsg := ' ';
			   BeamDiameterMsg := ' ';
			   WavelengthRangeMsg := ' ';				   	 
  			   SensorTypeMsg := ' ';
			   CalibMsg := ' ';
			   _itemRaisedProperties := 10;																																								
				
			10: GetCalibConfig();
				_itemRaisedProperties := 11;							
		
			11:  _pulseGeneratorMsg(IN := TRUE, PT := T#90MS); // 40MS + 10MS de temps de cycle = 50 MS 
				IF _pulseGeneratorMsg.Q THEN
					_pulseGeneratorMsg(IN := FALSE);
								
					GetResponsivity();							
					_itemScheduler := 50;
				END_IF
				
			(* Not necessary *)
			(*
			10: GetIdentifier();
				_itemRaisedProperties := 11;
				
			11: GetSensorType();
				_itemRaisedProperties := 12;
			
			12: GetWavelength();
				_itemRaisedProperties := 13;	

			12: GetBeamDiameter();
				_itemRaisedProperties := 16;
	
			13: GetWavelengthRange();
				_itemRaisedProperties := 16;
	
			14:  GetMaxPower();
				_itemRaisedProperties := 15;
				
			15: GetMinPower();
				_itemRaisedProperties := 16;
				
			17: GetSensorAttenuation();
				_itemRaisedProperties := 19;*)
				
			50: 
				_logger.Information(_message.Reset().
								    Append(Conf.Name).
								    Append(' - RaisePropertiesChanged').ToString());
				_raiseProperties := FALSE;				
				_itemRaisedProperties := 0;
		
		END_CASE	
	ELSE
		_pulseGenerator(IN := TRUE, PT := T#100MS);	
	END_IF
END_IF

*)
END_METHOD

{attribute 'TcRpcEnable' := '1'}
METHOD RangesVariation
VAR_INPUT
	Execute : BOOL;
	RangeValue : STRING;
END_VAR
VAR
	cmd : STRING := 'Sense:Power:Dc:Range:UPPer ';
END_VAR
IF Execute THEN
	_logger.Information(_message.Reset().
								Append(Conf.Name).
								Append(' - Set the range').ToString());
	
	Abort(_abortCmd);
	SerialCom.Send(CONCAT(cmd, TO_STRING(RangeValue)));	
	_rangeVariation := FALSE;
END_IF
END_METHOD

(** Read measure current **)
METHOD ReadCurrent
VAR_INPUT
END_VAR
VAR	
	cmd : STRING := 'Measure:Scalar:CURRent?';	
END_VAR
_deliverMessages := EFeedbackMsgPM101.CurrentMsg;
SerialCom.Send(cmd);
END_METHOD

(** Read measure power **)
METHOD ReadPower	
VAR_INPUT
END_VAR
VAR	
	cmd : STRING := 'Measure:Scalar:POWer?';	
END_VAR
_deliverMessages := EFeedbackMsgPM101.PowerMsg;
SerialCom.Send(cmd);
END_METHOD

{attribute 'TcRpcEnable' := '1'}
(** Sets the beam diameter in mm **)
METHOD SetBeamDiameter
VAR_INPUT
	Execute : BOOL;
	BeamDiameterValue : UINT;
END_VAR
VAR
	cmd : STRING := 'Sense:Correction:beamdiameter ';
END_VAR
IF Execute AND _pulseGeneratorCmd.Q THEN
	_logger.Information(_message.Reset().
								Append(Conf.Name).
								Append(' - Sets the beam diameter').ToString());
	
	SerialCom.Send(CONCAT(cmd, TO_STRING(BeamDiameterValue)));		
END_IF

IF Execute THEN
	IF _pulseGeneratorCmd.Q THEN
		_pulseGeneratorCmd(IN := FALSE, PT := T#10MS);									
		_setBeamDiameter := FALSE;
	ELSE
		_pulseGeneratorCmd(IN := Execute, PT := T#100MS);										
	END_IF
END_IF
END_METHOD

{attribute 'TcRpcEnable' := '1'}
(** Sets the responsivity mA/W **)
METHOD SetResponsivity
VAR_INPUT
	Execute : BOOL;
	ResponsivityValue : LREAL;
END_VAR
VAR
	cmd : STRING := 'SENSe:CORRection:POWer:PDIode ';
	setpoint : LREAL;	
END_VAR
IF Execute THEN			
	_monitoringMessages := FALSE;		
	_setResponsivity := TRUE;	
	_setpoint := ResponsivityValue;	
	
	CASE _itemExecScheduler OF
		0: _logger.Information(_message.Reset().
								Append(Conf.Name).
								Append(' - Set the responsivity: ').
								Append(TO_STRING(_setpoint)).ToString());	
			
			_abortCmd := TRUE;
			_itemExecScheduler := 1;			
			
		1:	IF NOT _abortCmd THEN
				_itemExecScheduler := 2;	
			END_IF						
						
  	   	2:	_logger.Information(_message.Reset().Append(Conf.Name).Append(' - Send setpoint').ToString());
			setpoint := _setpoint / 1000;
			SerialCom.Send(CONCAT(cmd, TO_STRING(setpoint)));										
			_itemExecScheduler := 3;				         					
			 	
		3:  _logger.Information(_message.Reset().Append(Conf.Name).Append(' - Get responsivity').ToString());
			GetResponsivity();
			_itemExecScheduler := 10;		 						

		4:  IF message = ' ' THEN
				_itemExecScheduler := 10;
			END_IF				

		10: _logger.Information(_message.Reset().Append(Conf.Name).Append(' - Done responsivity').ToString());
			_setpoint := 0;
			_setResponsivity := FALSE;	
			_itemExecScheduler := 0;	

			_monitoringMessages := TRUE;								
	END_CASE	
END_IF


(*1: _execPulseGenerator(IN := TRUE, PT := T#50MS);
			IF _execPulseGenerator.Q THEN
				_execPulseGenerator(IN := FALSE);
				_logger.Information(_message.Reset().Append(Conf.Name).Append(' - GetResponsivity').ToString());

				GetResponsivity();
				_itemExecScheduler := 2;		
			END_IF
		*)	

(*
IF Execute THEN	
	_setResponsivity := TRUE;	
	_setpoint := ResponsivityValue;	
	
	CASE _itemExecScheduler OF
		0: _logger.Information(_message.Reset().
								Append(Conf.Name).
								Append(' - Set the responsivity: ').
								Append(TO_STRING(_setpoint)).ToString());	

			setpoint := _setpoint / 1000;
			SerialCom.Send(CONCAT(cmd, TO_STRING(setpoint)));										
			_itemExecScheduler := 1;				
        
		1:	_execPulseGenerator(IN := TRUE, PT := wait1);
			IF _execPulseGenerator.Q THEN
				_execPulseGenerator(IN := FALSE);
				_logger.Information(_message.Reset().Append(Conf.Name).Append(' - Wait Set Responsivity: ').ToString());								    				
				_itemExecScheduler := 2;
			END_IF
					
			GetResponsivity();
			_itemExecScheduler := 3;
		
		3:  _execPulseGenerator(IN := TRUE, PT := wait2);
			IF _execPulseGenerator.Q THEN
				_execPulseGenerator(IN := FALSE);
				
				_logger.Information(_message.Reset().Append('Wait Get Responsivity').ToString());				
				_itemExecScheduler := 10;
			END_IF						
			
		10:  _setpoint := 0;
			_setResponsivity := FALSE;	
			_itemExecScheduler := 0;		
							
	END_CASE	
END_IF
*)

(*
IF Execute THEN	
	_setResponsivity := TRUE;	

	_setpoint := ResponsivityValue;
	
	IF _execPulseGenerator.Q THEN
		_execPulseGenerator(IN := FALSE);
			
		CASE _itemExecScheduler OF
			0: _logger.Information(_message.Reset().
									Append(Conf.Name).
									Append(' - Set the responsivity: ').
									Append(TO_STRING(_setpoint)).ToString());
				
				SerialCom.Send(CONCAT(cmd, TO_STRING(_setpoint / 1000)));
				_itemExecScheduler := 1;				

			1:  _itemExecScheduler := 2;

			2:  _itemExecScheduler := 3;
			
			3:  _itemExecScheduler := 4;
			
			4:  _itemExecScheduler := 5;			
	
			5:  GetResponsivity();
				_itemExecScheduler := 10;
				
			10:  _setpoint := 0;
				_setResponsivity := FALSE;	
				_itemExecScheduler := 0;		
								
		END_CASE
	ELSE
		_execPulseGenerator(IN := TRUE, PT := T#50MS);	
	END_IF
END_IF*)
END_METHOD

{attribute 'TcRpcEnable' := '1'}
(** Sets a user attenuation factor in dB **)
METHOD SetSensorAttenuation
VAR_INPUT
	Execute : BOOL;
	AttenuationValue : UINT;
END_VAR
VAR
	cmd : STRING := 'Sense:Correction:Loss:Input:MAGNitude ';
END_VAR
IF Execute AND _pulseGeneratorCmd.Q THEN
	_logger.Information(_message.Reset().
								Append(Conf.Name).
								Append(' - Sets a user attenuation factor').ToString());
	
	SerialCom.Send(CONCAT(cmd, TO_STRING(AttenuationValue)));		
END_IF

IF Execute THEN
	IF _pulseGeneratorCmd.Q THEN
		_pulseGeneratorCmd(IN := FALSE, PT := T#10MS);									
		_setSensorAttenuation := FALSE;
	ELSE
		_pulseGeneratorCmd(IN := Execute, PT := T#100MS);										
	END_IF
END_IF
END_METHOD

{attribute 'TcRpcEnable' := '1'}
(** Sets default sensor adapter type **)
METHOD SetSensorType
VAR_INPUT
	Execute : BOOL;
	SensorTypeValue : STRING;
END_VAR
VAR
	cmd : STRING := 'Input:Adapter:TYPE ';
END_VAR
IF Execute AND _pulseGeneratorCmd.Q THEN
	_logger.Information(_message.Reset().
								Append(Conf.Name).
								Append(' - Sets default sensor adapter type').ToString());
	
	SerialCom.Send(CONCAT(cmd, SensorTypeValue));		
END_IF

IF Execute THEN
	IF _pulseGeneratorCmd.Q THEN
		_pulseGeneratorCmd(IN := FALSE, PT := T#10MS);									
		_setSensorType := FALSE;
	ELSE
		_pulseGeneratorCmd(IN := Execute, PT := T#100MS);										
	END_IF	
END_IF
END_METHOD

{attribute 'TcRpcEnable' := '1'}
(** Sets the operation wavelength in nm **)
METHOD SetWavelength
VAR_INPUT
	Execute : BOOL;
	WavelengthValue : UINT;
END_VAR
VAR
	cmd : STRING := 'Sense:Correction:WAVelength ';
END_VAR
IF Execute AND _pulseGeneratorCmd.Q THEN
	_logger.Information(_message.Reset().
								Append(Conf.Name).
								Append(' - Sets the operation wavelength').ToString());
	
	SerialCom.Send(CONCAT(cmd, TO_STRING(WavelengthValue)));		
END_IF

IF Execute THEN
	IF _pulseGeneratorCmd.Q THEN
		_pulseGeneratorCmd(IN := FALSE, PT := T#10MS);									
		_setWavelength := FALSE;
	ELSE
		_pulseGeneratorCmd(IN := Execute, PT := T#100MS);										
	END_IF
END_IF
END_METHOD

METHOD SlowMessageScheduler
VAR_INPUT
END_VAR
IF _pulseGeneratorMsg.Q THEN
	_pulseGeneratorMsg(IN := FALSE, PT := T#10MS);
		
	CASE _itemScheduler OF
		0:	ReadPower();
			_itemScheduler := 2;						
	
		1: GetResponsivity();
			_itemScheduler := 0;			
			
		2 : GetDarkAdjustState();
			_itemScheduler := 3;		
	
		3 : GetDarkOffset();
			_itemScheduler := 0;

		4:  ReadCurrent();
			_itemScheduler := 0;			
		
	END_CASE
ELSE
	_pulseGeneratorMsg(IN := TRUE, PT := T#50MS);	
END_IF
END_METHOD

{attribute 'TcRpcEnable' := '1'}
(** Start dark adjust **)
METHOD StartDarkAdjust
VAR_INPUT
	Execute : BOOL;
END_VAR
VAR	
	cmd : STRING := 'Sense:CORRection:COLLect:ZERO:INITiate';	
END_VAR
IF Execute THEN	
	_startDarkAdjust := TRUE;	
	
	IF _execPulseGenerator.Q THEN
		_execPulseGenerator(IN := FALSE);
			
		CASE _itemExecScheduler OF
			0: _logger.Information(_message.Reset().
									Append(Conf.Name).
									Append(' - Start dark adjust').ToString());
				
				_darkOffset_mW := 0;
				SerialCom.Send(cmd);
				_itemExecScheduler := 1;				
				
			1:  GetDarkOffset();
				_itemExecScheduler := 2;
				
			2:  IF _darkOffset_mW = 0 THEN
					_logger.Information(_message.Reset().
									Append(Conf.Name).
									Append(' - Retry start dark adjust').ToString());
					_itemExecScheduler := 0;
				ELSE
					_itemExecScheduler := 10;
				END_IF
				
			10: _startDarkAdjust := FALSE;	
				_itemExecScheduler := 0;		
								
		END_CASE
	ELSE
		_execPulseGenerator(IN := TRUE, PT := T#80MS);	
	END_IF
END_IF
END_METHOD

END_FUNCTION_BLOCK

// ---- PMShared/Hardware/Devices/OpticalPowermeters/OpticalPowermeterBase.TcPOU
FUNCTION_BLOCK ABSTRACT OpticalPowermeterBase EXTENDS TExecution IMPLEMENTS IDevice
VAR_INPUT
END_VAR
VAR_OUTPUT
END_VAR
VAR
	{attribute 'OPC.UA.DA' := '0'}
	_name : STRING;
	{attribute 'OPC.UA.DA' := '0'}
	_deviceID : STRING;					
	{attribute 'OPC.UA.DA' := '0'}
	_family : DeviceFamily;	
	{attribute 'OPC.UA.DA' := '0'}
	_logger : Logger;
	{attribute 'OPC.UA.DA' := '0'}
	_message : StringBuilder;
	{attribute 'OPC.UA.DA' := '0'}
	_opticalPowermeterConfig : DeviceConfiguration;	
END_VAR

PROPERTY DeviceID : STRING
GET
DeviceID := _deviceID;
END_GET
SET
_deviceID := DeviceID;
END_SET
END_PROPERTY

PROPERTY Family : DeviceFamily
GET
Family := _family;
END_GET
SET
_family := Family;
END_SET
END_PROPERTY

PROPERTY Name : STRING
GET
Name := _name;
END_GET
SET
_name := Name;
END_SET
END_PROPERTY

END_FUNCTION_BLOCK

// ---- PMShared/Hardware/Devices/OpticalPowermeters/Thorlabs/PM101/PM101OpticalPowermeterHt.TcPOU
{attribute 'OPC.UA.DA' := '1'}
FUNCTION_BLOCK PM101OpticalPowermeterHt EXTENDS PM101OpticalPowermeter
VAR_INPUT
END_VAR
VAR_OUTPUT
END_VAR
VAR
	{attribute 'OPC.UA.DA' := '0'}
	_config : PM101OpticalPowermeterConfig;
	{attribute 'OPC.UA.DA' := '0'}
	_polarisationConfig : PolarisationConfig;
	{attribute 'OPC.UA.DA' := '0'}
	_rFactorSettings : RFactorSettings;
	{attribute 'OPC.UA.DA' := '0'}
	_responsivityConfig : ResponsivityConfig;
	{attribute 'OPC.UA.DA' := '0'}
	_coeAccess : CoeAccess;
	{attribute 'OPC.UA.DA' := '0'}
	_initConfigSerialCom : BOOL;
	{attribute 'OPC.UA.DA' := '0'}	
	_serialCom  : SerialCom(Prefix :='', Suffix := Const.LINE_FEED);
	{attribute 'OPC.UA.DA' := '0'}
	_refSerialCom : REFERENCE TO SerialCom(Prefix :='', Suffix := Const.LINE_FEEL) := _serialCom;
	
	{attribute 'OPC.UA.DA' := '0'}
	_pulseGeneratorInit : TON;	
	{attribute 'OPC.UA.DA' := '0'}
	_itemInit : INT;
END_VAR

IF _config.IsSimulated THEN
	SUPER^(Conf := _config, PolarisationConfig := _polarisationConfig, RFactorSettings := _rfactorSettings, ResponsivityConfig := _responsivityConfig, SerialCom := _serialCom, RefSerialCom := _refSerialCom);
ELSE
	IF NOT InitConfigSerialCom THEN
		ConfigureSerialCom();
	ELSIF THIS^.Status = TExecutionState.Ready THEN
		IF _refSerialCom.ErrorReceiveId = COMERROR_NOERROR THEN
			_refSerialCom(TxBuffer:= HardwareGlobalVariables.TxBufferOpticalPowermeterHt, 
						  RxBuffer:= HardwareGlobalVariables.RxBufferOpticalPowermeterHt);
		END_IF	
					
		// Init device
		InitDevice(); 
  
		SUPER^(Conf := _config, PolarisationConfig := _polarisationConfig, RFactorSettings := _rfactorSettings, ResponsivityConfig := _responsivityConfig, SerialCom := _serialCom, RefSerialCom := _refSerialCom);							
	END_IF
END_IF

METHOD ConfigureSerialCom
VAR_INPUT
END_VAR
IF _coeAccess.CoeOperation.Ready THEN
	_logger.Information(_message.Reset().Append('Start configuration com serial').ToString());
END_IF;	

_coeAccess.CoeOperation.Start();
_coeAccess(SerialCommunication := _config.SerialCommunication);
	
IF _coeAccess.CoeOperation.Done THEN
	_coeAccess.SetDone();
	
	_Logger.Information(_message.Reset().
							Append('{').Append(TO_STRING(THIS^.Family)).Append('} : ').
							Append(' - Status : ').Append(TO_STRING(_coeAccess.Status)).ToString());
	InitConfigSerialCom := TRUE;
END_IF
 
IF _coeAccess.CoeOperation.Error THEN	
	_coeAccess.SetError(0);
	
	_Logger.Error(_message.Reset().
							Append('{').Append(TO_STRING(THIS^.Family)).Append('} : ').
							Append(' - Status : ').Append(TO_STRING(_coeAccess.Status)).ToString());
	InitConfigSerialCom := TRUE;
END_IF

THIS^.Status := _coeAccess.Status;
State := _coeAccess.Status;
END_METHOD

METHOD FB_init : BOOL
VAR_INPUT
	bInitRetains : BOOL; // if TRUE, the retain variables are initialized (warm start / cold start)
	bInCopyCode : BOOL;  // if TRUE, the instance afterwards gets moved into the copy code (online change)
	Config : PM101OpticalPowermeterConfig;
	PolarisationConfig : PolarisationConfig;
	RFactorSettings : RFactorSettings;
	ResponsivityConfig : ResponsivityConfig;
END_VAR
IF Config.IsEnabled THEN
	_config := Config;
	_polarisationConfig := PolarisationConfig;
	_rFactorSettings := RFactorSettings;
	_responsivityConfig := ResponsivityConfig;
	
	SUPER^._opticalPowermeterConfig.Name := Config.Name;
	SUPER^._opticalPowermeterConfig.DeviceID := Config.DeviceID;
	SUPER^._opticalPowermeterConfig.IsEnabled := Config.IsEnabled;
	SUPER^._opticalPowermeterConfig.LogLevel := Config.LogLevel;
	
	SUPER^.Name := Config.Name;
	SUPER^.DeviceID := Config.DeviceID;	
	THIS^.Family := DeviceFamily.OpticalPowermeter;
		
	_Logger.Information(_message.Reset().Append('Init ').
							Append('{').Append(TO_STRING(THIS^.Family)).Append('} - ').
							Append('{').Append(TO_STRING(Config.Name)).Append('}').ToString());																													
END_IF
END_METHOD

PROPERTY InitConfigSerialCom : BOOL
GET
InitConfigSerialCom := _initConfigSerialCom;
END_GET
SET
_initConfigSerialCom := InitConfigSerialCom;
END_SET
END_PROPERTY

METHOD InitDevice 
VAR_INPUT	
END_VAR
IF NOT _initDevice THEN	
	CASE _itemInit OF
		0:  _logger.Information(_message.Reset().Append(_config.Name).Append(' - InitDevice').ToString());
			_itemInit := 1;
		
		1:  SUPER^._rangeAuto := TRUE;
			SUPER^._cmdRange := 'TRUE';
			_itemInit := 2;			
			
		2:  SUPER^._setSensorAttenuation := TRUE;
			SUPER^._cmdSensorAttenuation := _config.Sensor.Attenuation;
			_itemInit := 3;
			
		3:  IF _config.Sensor.Name = Const.POWERMETER_SENSOR_NAME_S150C THEN
				_logger.Error(_message.Reset().Append(_config.Name).Append(' - Sensor name: ').Append(_config.Sensor.Name).ToString());
				_itemInit := 10;
			ELSIF _config.Sensor.Name = Const.POWERMETER_SENSOR_NAME_TAP_COUPLER THEN
				_logger.Error(_message.Reset().Append(_config.Name).Append(' - Sensor name: ').Append(_config.Sensor.Name).ToString());
				_itemInit := 20;
			ELSE
				_logger.Error(_message.Reset().Append(_config.Name).Append(' - NAME OF FAILED SENSOR').ToString());
		    END_IF
			
		10:  SUPER^._setWavelength := TRUE;
			 SUPER^._cmdWavelength := _config.Sensor.Wavelength;
			 _itemInit := 50;		
		
		20:  GetResponsivity();
			 _itemInit := 21;
			
		21:	 _pulseGeneratorInit(IN := TRUE, PT := T#3000MS);
			 IF _pulseGeneratorInit.Q THEN
				_pulseGeneratorInit(IN := FALSE);				
			 	_itemInit := 22;
			 END_IF
		
		22:	 IF ResponsivityMsg = LREAL_TO_STRING(_responsivityConfig.Responsivity_mA_W) THEN
			 	_logger.Information(_message.Reset().Append(_config.Name).Append(' - Responsivity already defined').ToString());
			 	_itemInit := 50;
			 ELSE				 
				_itemInit := 23;
			 END_IF	
			 
		23:  _logger.Information(_message.Reset().
							Append(_config.Name).
							Append(' - Init responsivity: ').
							Append(LREAL_TO_STRING(_responsivityConfig.Responsivity_mA_W)).ToString());
			
			SUPER^._setpoint := _responsivityConfig.Responsivity_ma_W;
			SUPER^._setResponsivity := TRUE;
			
			_itemInit := 50;

		50: _logger.Information(_message.Reset().
							Append(_config.Name).
							Append(' - InitDevice done').ToString());				
			_initDevice	:= TRUE;
	END_CASE			
END_IF
END_METHOD

END_FUNCTION_BLOCK

// ---- PMShared/Hardware/Devices/DistanceSensors/MicroEpsilon/MicroEpsilonDistanceSensor.TcPOU
{attribute 'OPC.UA.DA' := '1'}
FUNCTION_BLOCK MicroEpsilonDistanceSensor EXTENDS DistanceSensorBase
VAR_INPUT
END_VAR
VAR_OUTPUT
END_VAR
VAR
	{attribute 'OPC.UA.DA' := '0'}
	_config : MicroEpsilonDistanceSensorConfig;
	{attribute 'OPC.UA.DA' := '0'}
	IoMicroEpsilonDistanceSensor : IoMicroEpsilonDistanceSensor;
	
	{attribute 'OPC.UA.DA' := '0'}
	_deliverMessages : INT;
	
	DistanceMsg : STRING(255);	
	IdMsg : STRING(255);
	CustomMsg : STRING(255);
	
	{region 'Commands'}
	
	{attribute 'OPC.UA.DA' := '0'}	
	_customCmd : BOOL;	
			  		   
	{endregion}
	
	{attribute 'OPC.UA.DA' := '0'}
	_initDevice : BOOL;	

	{attribute 'OPC.UA.DA' := '0'}
	_itemScheduler : INT;		
	{attribute 'OPC.UA.DA' := '0'}
	_pulseGenerator : TON;		 			
END_VAR


// Init device
InitDevice();

MessageScheduler();

METHOD FB_init : BOOL
VAR_INPUT
	bInitRetains : BOOL; // if TRUE, the retain variables are initialized (warm start / cold start)
	bInCopyCode : BOOL;  // if TRUE, the instance afterwards gets moved into the copy code (online change)
	Config : MicroEpsilonDistanceSensorConfig;
END_VAR
IF Config.IsEnabled THEN
	_config := Config;
	
	SUPER^._distanceSensorConfig.Name := Config.Name;
	SUPER^._distanceSensorConfig.DeviceID := Config.DeviceID;
	SUPER^._distanceSensorConfig.IsEnabled := Config.IsEnabled;
	SUPER^._distanceSensorConfig.LogLevel := Config.LogLevel;
	
	SUPER^.Name := Config.Name;
	SUPER^.DeviceID := Config.DeviceID;	
	THIS^.Family := DeviceFamily.DistanceSensors;
		
	_Logger.Information(_message.Reset().Append('Init ').
							Append('{').Append(TO_STRING(THIS^.Family)).Append('} - ').
							Append('{').Append(TO_STRING(Config.Name)).Append('}').ToString());																													
END_IF
END_METHOD

METHOD InitDevice
VAR_INPUT
END_VAR
IF NOT _initDevice THEN	
	_logger.Information(_message.Reset().Append(_config.Name).Append(' - Init device').ToString());

	THIS^.SetDone();							
	_initDevice := TRUE;	
END_IF
END_METHOD

METHOD MessageScheduler
VAR_INPUT
END_VAR
VAR
	distanceToMM : LREAL;
END_VAR
IF _pulseGenerator.Q THEN
	_pulseGenerator(IN := FALSE, PT := T#10MS);
		
	CASE _itemScheduler OF
		0:  			
			// The return value is in millimeter 
			//distanceToMM := TO_LREAL(IoMicroEpsilonDistanceSensor.InputMicroEpsilonDistanceSensor) / TO_LREAL(1000000);
			//DistanceMsg := LREAL_TO_STRING(distanceToMM);
			
			DistanceMsg := REAL_TO_STRING(IoMicroEpsilonDistanceSensor.InputMicroEpsilonDistanceSensor);
			_itemScheduler := 0;
					
